LIN {X 0,Y 211.317,Z 790.887,A -85,B 0,C 180,E1 4630.049,E2 4630.049} C_VEL
LIN {X 0,Y 204.375,Z 802.097,A -85,B 0,C 180,E1 4624.722,E2 4624.722} C_VEL
LIN {X 0,Y 199.04,Z 811.282,A -85,B 0,C 180,E1 4619.061,E2 4619.061} C_VEL
LIN {X 0,Y 195.25,Z 818.98,A -85,B 0,C 180,E1 4612.9,E2 4612.9} C_VEL
LIN {X 0,Y 193.221,Z 824.706,A -85,B 0,C 180,E1 4606.795,E2 4606.795} C_VEL
LIN {X 0,Y 192.563,Z 828.46,A -85,B 0,C 180,E1 4601.073,E2 4601.073} C_VEL
LIN {X 0,Y 192.668,Z 830.823,A -85,B 0,C 180,E1 4595.357,E2 4595.357} C_VEL
LIN {X 0,Y 192.832,Z 831.611,A -85,B 0,C 180,E1 4590.591,E2 4590.591} C_VEL
LIN {X 0,Y 192.717,Z 831.408,A -85,B 0,C 180,E1 4586.13,E2 4586.13} C_VEL
LIN {X 0,Y 192.494,Z 830.016,A -85,B 0,C 180,E1 4580.727,E2 4580.727} C_VEL
LIN {X 0,Y 192.901,Z 826.886,A -85,B 0,C 180,E1 4574.669,E2 4574.669} C_VEL
LIN {X 0,Y 194.828,Z 821.744,A -85,B 0,C 180,E1 4567.995,E2 4567.995} C_VEL
LIN {X 0,Y 198.485,Z 815.132,A -85,B 0,C 180,E1 4561.734,E2 4561.734} C_VEL
LIN {X 0,Y 204.073,Z 806.598,A -85,B 0,C 180,E1 4555.703,E2 4555.703} C_VEL
LIN {X 0,Y 211.205,Z 796.698,A -85,B 0,C 180,E1 4550.272,E2 4550.272} C_VEL
LIN {X 0,Y 220.022,Z 784.872,A -85,B 0,C 180,E1 4545.218,E2 4545.218} C_VEL
LIN {X 0,Y 229.843,Z 771.631,A -85,B 0,C 180,E1 4540.802,E2 4540.802} C_VEL
LIN {X 0,Y 240.325,Z 756.815,A -85,B 0,C 180,E1 4536.981,E2 4536.981} C_VEL
LIN {X 0,Y 250.499,Z 741.511,A -85,B 0,C 180,E1 4533.875,E2 4533.875} C_VEL
LIN {X 0,Y 261.006,Z 724.467,A -85,B 0,C 180,E1 4531.143,E2 4531.143} C_VEL
LIN {X 0,Y 270.771,Z 707,A -85,B 0,C 180,E1 4528.931,E2 4528.931} C_VEL
LIN {X 0,Y 280.133,Z 688.021,A -85,B 0,C 180,E1 4527.058,E2 4527.058} C_VEL
LIN {X 0,Y 288.655,Z 668.181,A -85,B 0,C 180,E1 4525.53,E2 4525.53} C_VEL
LIN {X 0,Y 296.228,Z 647.353,A -85,B 0,C 180,E1 4524.307,E2 4524.307} C_VEL
LIN {X 0,Y 302.485,Z 626.505,A -85,B 0,C 180,E1 4523.392,E2 4523.392} C_VEL
LIN {X 0,Y 307.54,Z 604.237,A -85,B 0,C 180,E1 4522.67,E2 4522.67} C_VEL
LIN {X 0,Y 310.852,Z 582.325,A -85,B 0,C 180,E1 4522.123,E2 4522.123} C_VEL
LIN {X 0,Y 326.311,Z 437.595,A -85,B 0,C 180,E1 4519.094,E2 4519.094} C_VEL
LIN {X 0,Y 324.635,Z 433.151,A -85,B 0,C 180,E1 4517.015,E2 4517.015} C_VEL
LIN {X 0,Y 323.554,Z 430.422,A -85,B 0,C 180,E1 4515.23,E2 4515.23} C_VEL
LIN {X 0,Y 322.63,Z 427.763,A -85,B 0,C 180,E1 4512.712,E2 4512.712} C_VEL
LIN {X 0,Y 322.365,Z 427.503,A -85,B 0,C 180,E1 4509.103,E2 4509.103} C_VEL
LIN {X 0,Y 322.631,Z 428.25,A -85,B 0,C 180,E1 4507.749,E2 4507.749} C_VEL
LIN {X 0,Y 323.747,Z 431.704,A -85,B 0,C 180,E1 4504.873,E2 4504.873} C_VEL
LIN {X 0,Y 325.23,Z 435.825,A -85,B 0,C 180,E1 4502.645,E2 4502.645} C_VEL
LIN {X 0,Y 325.665,Z 437.428,A -85,B 0,C 180,E1 4502.072,E2 4502.072} C_VEL
LIN {X 0,Y 308.977,Z 582.418,A -85,B 0,C 180,E1 4499.021,E2 4499.021} C_VEL
LIN {X 0,Y 305.09,Z 603.307,A -85,B 0,C 180,E1 4498.354,E2 4498.354} C_VEL
LIN {X 0,Y 300.007,Z 623.447,A -85,B 0,C 180,E1 4497.469,E2 4497.469} C_VEL
LIN {X 0,Y 293.506,Z 643.814,A -85,B 0,C 180,E1 4496.291,E2 4496.291} C_VEL
LIN {X 0,Y 286.577,Z 661.874,A -85,B 0,C 180,E1 4494.957,E2 4494.957} C_VEL
LIN {X 0,Y 278.381,Z 679.801,A -85,B 0,C 180,E1 4493.278,E2 4493.278} C_VEL
LIN {X 0,Y 269.137,Z 697.434,A -85,B 0,C 180,E1 4491.201,E2 4491.201} C_VEL
LIN {X 0,Y 259.035,Z 714.421,A -85,B 0,C 180,E1 4488.653,E2 4488.653} C_VEL
LIN {X 0,Y 249.221,Z 729.24,A -85,B 0,C 180,E1 4485.836,E2 4485.836} C_VEL
LIN {X 0,Y 239.085,Z 743.194,A -85,B 0,C 180,E1 4482.465,E2 4482.465} C_VEL
LIN {X 0,Y 228.642,Z 756.385,A -85,B 0,C 180,E1 4478.327,E2 4478.327} C_VEL
LIN {X 0,Y 219.438,Z 767.23,A -85,B 0,C 180,E1 4473.852,E2 4473.852} C_VEL
LIN {X 0,Y 211.365,Z 776.379,A -85,B 0,C 180,E1 4468.899,E2 4468.899} C_VEL
LIN {X 0,Y 204.471,Z 784.06,A -85,B 0,C 180,E1 4463.321,E2 4463.321} C_VEL
LIN {X 0,Y 199.247,Z 789.969,A -85,B 0,C 180,E1 4457.359,E2 4457.359} C_VEL
LIN {X 0,Y 195.774,Z 794.085,A -85,B 0,C 180,E1 4451.214,E2 4451.214} C_VEL
LIN {X 0,Y 193.917,Z 796.385,A -85,B 0,C 180,E1 4445.277,E2 4445.277} C_VEL
LIN {X 0,Y 193.148,Z 797.233,A -85,B 0,C 180,E1 4439.461,E2 4439.461} C_VEL
LIN {X 0,Y 193.025,Z 796.836,A -85,B 0,C 180,E1 4433.834,E2 4433.834} C_VEL
LIN {X 0,Y 193.474,Z 794.978,A -85,B 0,C 180,E1 4428.041,E2 4428.041} C_VEL
LIN {X 0,Y 194.932,Z 791.439,A -85,B 0,C 180,E1 4421.843,E2 4421.843} C_VEL
LIN {X 0,Y 197.726,Z 786.247,A -85,B 0,C 180,E1 4415.808,E2 4415.808} C_VEL
LIN {X 0,Y 201.96,Z 779.409,A -85,B 0,C 180,E1 4410.063,E2 4410.063} C_VEL
LIN {X 0,Y 207.83,Z 770.496,A -85,B 0,C 180,E1 4404.481,E2 4404.481} C_VEL
LIN {X 0,Y 214.723,Z 760.117,A -85,B 0,C 180,E1 4399.54,E2 4399.54} C_VEL
LIN {X 0,Y 222.414,Z 748.305,A -85,B 0,C 180,E1 4395.156,E2 4395.156} C_VEL
LIN {X 0,Y 230.633,Z 735.088,A -85,B 0,C 180,E1 4391.291,E2 4391.291} C_VEL
LIN {X 0,Y 239.139,Z 720.459,A -85,B 0,C 180,E1 4387.898,E2 4387.898} C_VEL
LIN {X 0,Y 247.432,Z 704.923,A -85,B 0,C 180,E1 4385.024,E2 4385.024} C_VEL
LIN {X 0,Y 255.907,Z 687.184,A -85,B 0,C 180,E1 4382.423,E2 4382.423} C_VEL
LIN {X 0,Y 263.586,Z 668.825,A -85,B 0,C 180,E1 4380.298,E2 4380.298} C_VEL
LIN {X 0,Y 270.362,Z 650.051,A -85,B 0,C 180,E1 4378.573,E2 4378.573} C_VEL
LIN {X 0,Y 276.368,Z 630.229,A -85,B 0,C 180,E1 4377.137,E2 4377.137} C_VEL
LIN {X 0,Y 281.45,Z 609.5,A -85,B 0,C 180,E1 4375.988,E2 4375.988} C_VEL
LIN {X 0,Y 285.444,Z 588.089,A -85,B 0,C 180,E1 4375.117,E2 4375.117} C_VEL
LIN {X 0,Y 288.238,Z 565.56,A -85,B 0,C 180,E1 4374.491,E2 4374.491} C_VEL
LIN {X 0,Y 301.041,Z 423.363,A -85,B 0,C 180,E1 4371.364,E2 4371.364} C_VEL
LIN {X 0,Y 293.436,Z 409.422,A -85,B 0,C 180,E1 4367.547,E2 4367.547} C_VEL
LIN {X 0,Y 287.048,Z 398.81,A -85,B 0,C 180,E1 4363.864,E2 4363.864} C_VEL
LIN {X 0,Y 282.288,Z 391.221,A -85,B 0,C 180,E1 4360.669,E2 4360.669} C_VEL
LIN {X 0,Y 279.028,Z 386.353,A -85,B 0,C 180,E1 4358.177,E2 4358.177} C_VEL
LIN {X 0,Y 276.012,Z 381.873,A -85,B 0,C 180,E1 4355.547,E2 4355.547} C_VEL
LIN {X 0,Y 272.92,Z 377.285,A -85,B 0,C 180,E1 4352.333,E2 4352.333} C_VEL
LIN {X 0,Y 269.763,Z 372.7,A -85,B 0,C 180,E1 4348.078,E2 4348.078} C_VEL
LIN {X 0,Y 266.645,Z 368.098,A -85,B 0,C 180,E1 4340.637,E2 4340.637} C_VEL
LIN {X 0,Y 266.222,Z 367.692,A -85,B 0,C 180,E1 4334.572,E2 4334.572} C_VEL
LIN {X 0,Y 267.044,Z 368.731,A -85,B 0,C 180,E1 4330.57,E2 4330.57} C_VEL
LIN {X 0,Y 268.111,Z 370.684,A -85,B 0,C 180,E1 4327.627,E2 4327.627} C_VEL
LIN {X 0,Y 268.708,Z 372.408,A -85,B 0,C 180,E1 4326.259,E2 4326.259} C_VEL
LIN {X 0,Y 269.521,Z 377.466,A -85,B 0,C 180,E1 4324.137,E2 4324.137} C_VEL
LIN {X 0,Y 270.707,Z 383.214,A -85,B 0,C 180,E1 4321.82,E2 4321.82} C_VEL
LIN {X 0,Y 271.569,Z 384.888,A -85,B 0,C 180,E1 4320.705,E2 4320.705} C_VEL
LIN {X 0,Y 273.038,Z 386.963,A -85,B 0,C 180,E1 4319.065,E2 4319.065} C_VEL
LIN {X 0,Y 276.48,Z 392.054,A -85,B 0,C 180,E1 4315.747,E2 4315.747} C_VEL
LIN {X 0,Y 280.407,Z 397.981,A -85,B 0,C 180,E1 4312.572,E2 4312.572} C_VEL
LIN {X 0,Y 285.065,Z 405.319,A -85,B 0,C 180,E1 4309.336,E2 4309.336} C_VEL
LIN {X 0,Y 291.595,Z 415.977,A -85,B 0,C 180,E1 4305.452,E2 4305.452} C_VEL
LIN {X 0,Y 298.484,Z 428.22,A -85,B 0,C 180,E1 4301.898,E2 4301.898} C_VEL
LIN {X 0,Y 301.017,Z 433.158,A -85,B 0,C 180,E1 4300.693,E2 4300.693} C_VEL
LIN {X 0,Y 286.835,Z 594.303,A -85,B 0,C 180,E1 4297.252,E2 4297.252} C_VEL
LIN {X 0,Y 283.258,Z 616.443,A -85,B 0,C 180,E1 4296.578,E2 4296.578} C_VEL
LIN {X 0,Y 278.332,Z 637.822,A -85,B 0,C 180,E1 4295.714,E2 4295.714} C_VEL
LIN {X 0,Y 272.14,Z 659.139,A -85,B 0,C 180,E1 4294.54,E2 4294.54} C_VEL
LIN {X 0,Y 265.201,Z 679.03,A -85,B 0,C 180,E1 4293.099,E2 4293.099} C_VEL
LIN {X 0,Y 257.115,Z 698.659,A -85,B 0,C 180,E1 4291.266,E2 4291.266} C_VEL
LIN {X 0,Y 248.687,Z 716.603,A -85,B 0,C 180,E1 4289.13,E2 4289.13} C_VEL
LIN {X 0,Y 239.009,Z 735.048,A -85,B 0,C 180,E1 4286.349,E2 4286.349} C_VEL
LIN {X 0,Y 230.023,Z 750.696,A -85,B 0,C 180,E1 4283.358,E2 4283.358} C_VEL
LIN {X 0,Y 220.474,Z 766.1,A -85,B 0,C 180,E1 4279.626,E2 4279.626} C_VEL
LIN {X 0,Y 211.738,Z 779.481,A -85,B 0,C 180,E1 4275.478,E2 4275.478} C_VEL
LIN {X 0,Y 203.307,Z 792.156,A -85,B 0,C 180,E1 4270.475,E2 4270.475} C_VEL
LIN {X 0,Y 196.415,Z 802.743,A -85,B 0,C 180,E1 4265.112,E2 4265.112} C_VEL
LIN {X 0,Y 190.906,Z 811.872,A -85,B 0,C 180,E1 4259.145,E2 4259.145} C_VEL
LIN {X 0,Y 187.202,Z 819.025,A -85,B 0,C 180,E1 4252.944,E2 4252.944} C_VEL
LIN {X 0,Y 185.121,Z 824.711,A -85,B 0,C 180,E1 4246.308,E2 4246.308} C_VEL
LIN {X 0,Y 184.564,Z 828.324,A -85,B 0,C 180,E1 4240.295,E2 4240.295} C_VEL
LIN {X 0,Y 184.735,Z 830.276,A -85,B 0,C 180,E1 4234.653,E2 4234.653} C_VEL
LIN {X 0,Y 184.878,Z 830.91,A -85,B 0,C 180,E1 4229.997,E2 4229.997} C_VEL
LIN {X 0,Y 184.705,Z 830.615,A -85,B 0,C 180,E1 4225.339,E2 4225.339} C_VEL
LIN {X 0,Y 184.52,Z 828.929,A -85,B 0,C 180,E1 4219.38,E2 4219.38} C_VEL
LIN {X 0,Y 185.127,Z 825.839,A -85,B 0,C 180,E1 4213.363,E2 4213.363} C_VEL
LIN {X 0,Y 187.473,Z 820.555,A -85,B 0,C 180,E1 4206.418,E2 4206.418} C_VEL
LIN {X 0,Y 191.675,Z 813.79,A -85,B 0,C 180,E1 4199.945,E2 4199.945} C_VEL
LIN {X 0,Y 197.916,Z 805.198,A -85,B 0,C 180,E1 4193.763,E2 4193.763} C_VEL
LIN {X 0,Y 205.71,Z 795.146,A -85,B 0,C 180,E1 4188.246,E2 4188.246} C_VEL
LIN {X 0,Y 215.604,Z 782.696,A -85,B 0,C 180,E1 4182.979,E2 4182.979} C_VEL
LIN {X 0,Y 226.224,Z 769.059,A -85,B 0,C 180,E1 4178.551,E2 4178.551} C_VEL
LIN {X 0,Y 236.749,Z 754.9,A -85,B 0,C 180,E1 4174.98,E2 4174.98} C_VEL
LIN {X 0,Y 247.404,Z 739.443,A -85,B 0,C 180,E1 4171.926,E2 4171.926} C_VEL
LIN {X 0,Y 258.406,Z 722.059,A -85,B 0,C 180,E1 4169.242,E2 4169.242} C_VEL
LIN {X 0,Y 268.469,Z 704.499,A -85,B 0,C 180,E1 4167.11,E2 4167.11} C_VEL
LIN {X 0,Y 278.154,Z 685.338,A -85,B 0,C 180,E1 4165.301,E2 4165.301} C_VEL
LIN {X 0,Y 286.741,Z 665.592,A -85,B 0,C 180,E1 4163.86,E2 4163.86} C_VEL
LIN {X 0,Y 294.301,Z 645.023,A -85,B 0,C 180,E1 4162.718,E2 4162.718} C_VEL
LIN {X 0,Y 300.678,Z 623.698,A -85,B 0,C 180,E1 4161.842,E2 4161.842} C_VEL
LIN {X 0,Y 305.706,Z 601.598,A -85,B 0,C 180,E1 4161.161,E2 4161.161} C_VEL
LIN {X 0,Y 309.082,Z 578.98,A -85,B 0,C 180,E1 4160.621,E2 4160.621} C_VEL
LIN {X 0,Y 324.139,Z 443.084,A -85,B 0,C 180,E1 4157.844,E2 4157.844} C_VEL
LIN {X 0,Y 322.498,Z 438.528,A -85,B 0,C 180,E1 4155.281,E2 4155.281} C_VEL
LIN {X 0,Y 321.524,Z 435.658,A -85,B 0,C 180,E1 4152.574,E2 4152.574} C_VEL
LIN {X 0,Y 321.29,Z 435.43,A -85,B 0,C 180,E1 4149.134,E2 4149.134} C_VEL
LIN {X 0,Y 321.513,Z 436.195,A -85,B 0,C 180,E1 4147.866,E2 4147.866} C_VEL
LIN {X 0,Y 322.481,Z 439.462,A -85,B 0,C 180,E1 4145.16,E2 4145.16} C_VEL
LIN {X 0,Y 323.554,Z 442.72,A -85,B 0,C 180,E1 4143.358,E2 4143.358} C_VEL
LIN {X 0,Y 306.938,Z 582.808,A -85,B 0,C 180,E1 4140.461,E2 4140.461} C_VEL
LIN {X 0,Y 302.915,Z 603.797,A -85,B 0,C 180,E1 4139.806,E2 4139.806} C_VEL
LIN {X 0,Y 297.764,Z 623.721,A -85,B 0,C 180,E1 4138.954,E2 4138.954} C_VEL
LIN {X 0,Y 291.177,Z 643.893,A -85,B 0,C 180,E1 4137.82,E2 4137.82} C_VEL
LIN {X 0,Y 283.519,Z 663.131,A -85,B 0,C 180,E1 4136.423,E2 4136.423} C_VEL
LIN {X 0,Y 274.65,Z 681.852,A -85,B 0,C 180,E1 4134.684,E2 4134.684} C_VEL
LIN {X 0,Y 265.153,Z 699.145,A -85,B 0,C 180,E1 4132.643,E2 4132.643} C_VEL
LIN {X 0,Y 254.743,Z 715.871,A -85,B 0,C 180,E1 4130.129,E2 4130.129} C_VEL
LIN {X 0,Y 244.058,Z 731.223,A -85,B 0,C 180,E1 4127.18,E2 4127.18} C_VEL
LIN {X 0,Y 233.712,Z 744.734,A -85,B 0,C 180,E1 4123.857,E2 4123.857} C_VEL
LIN {X 0,Y 223.496,Z 757.002,A -85,B 0,C 180,E1 4119.971,E2 4119.971} C_VEL
LIN {X 0,Y 213.636,Z 768.004,A -85,B 0,C 180,E1 4115.387,E2 4115.387} C_VEL
LIN {X 0,Y 205.343,Z 776.816,A -85,B 0,C 180,E1 4110.545,E2 4110.545} C_VEL
LIN {X 0,Y 197.578,Z 784.879,A -85,B 0,C 180,E1 4104.567,E2 4104.567} C_VEL
LIN {X 0,Y 192.047,Z 790.635,A -85,B 0,C 180,E1 4098.569,E2 4098.569} C_VEL
LIN {X 0,Y 188.135,Z 794.847,A -85,B 0,C 180,E1 4092.043,E2 4092.043} C_VEL
LIN {X 0,Y 186.051,Z 797.16,A -85,B 0,C 180,E1 4085.764,E2 4085.764} C_VEL
LIN {X 0,Y 185.192,Z 797.967,A -85,B 0,C 180,E1 4079.636,E2 4079.636} C_VEL
LIN {X 0,Y 185.054,Z 797.56,A -85,B 0,C 180,E1 4073.909,E2 4073.909} C_VEL
LIN {X 0,Y 185.522,Z 795.705,A -85,B 0,C 180,E1 4067.894,E2 4067.894} C_VEL
LIN {X 0,Y 186.973,Z 792.374,A -85,B 0,C 180,E1 4061.728,E2 4061.728} C_VEL
LIN {X 0,Y 189.7,Z 787.592,A -85,B 0,C 180,E1 4055.751,E2 4055.751} C_VEL
LIN {X 0,Y 194.088,Z 780.826,A -85,B 0,C 180,E1 4049.708,E2 4049.708} C_VEL
LIN {X 0,Y 199.732,Z 772.618,A -85,B 0,C 180,E1 4044.257,E2 4044.257} C_VEL
LIN {X 0,Y 206.772,Z 762.571,A -85,B 0,C 180,E1 4039.133,E2 4039.133} C_VEL
LIN {X 0,Y 215.113,Z 750.424,A -85,B 0,C 180,E1 4034.363,E2 4034.363} C_VEL
LIN {X 0,Y 223.579,Z 737.487,A -85,B 0,C 180,E1 4030.406,E2 4030.406} C_VEL
LIN {X 0,Y 232.336,Z 723.177,A -85,B 0,C 180,E1 4026.948,E2 4026.948} C_VEL
LIN {X 0,Y 241.451,Z 706.786,A -85,B 0,C 180,E1 4023.834,E2 4023.834} C_VEL
LIN {X 0,Y 249.848,Z 689.894,A -85,B 0,C 180,E1 4021.303,E2 4021.303} C_VEL
LIN {X 0,Y 257.65,Z 672.182,A -85,B 0,C 180,E1 4019.189,E2 4019.189} C_VEL
LIN {X 0,Y 265.031,Z 652.803,A -85,B 0,C 180,E1 4017.355,E2 4017.355} C_VEL
LIN {X 0,Y 271.202,Z 633.569,A -85,B 0,C 180,E1 4015.92,E2 4015.92} C_VEL
LIN {X 0,Y 276.606,Z 612.831,A -85,B 0,C 180,E1 4014.731,E2 4014.731} C_VEL
LIN {X 0,Y 280.958,Z 590.736,A -85,B 0,C 180,E1 4013.808,E2 4013.808} C_VEL
LIN {X 0,Y 283.853,Z 569.055,A -85,B 0,C 180,E1 4013.186,E2 4013.186} C_VEL
LIN {X 0,Y 297.056,Z 427.726,A -85,B 0,C 180,E1 4010.119,E2 4010.119} C_VEL
LIN {X 0,Y 290.081,Z 414.776,A -85,B 0,C 180,E1 4006.424,E2 4006.424} C_VEL
LIN {X 0,Y 283.791,Z 404.153,A -85,B 0,C 180,E1 4002.564,E2 4002.564} C_VEL
LIN {X 0,Y 278.928,Z 396.293,A -85,B 0,C 180,E1 3999.041,E2 3999.041} C_VEL
LIN {X 0,Y 274.567,Z 389.623,A -85,B 0,C 180,E1 3995.25,E2 3995.25} C_VEL
LIN {X 0,Y 271.442,Z 384.916,A -85,B 0,C 180,E1 3991.907,E2 3991.907} C_VEL
LIN {X 0,Y 268.47,Z 380.465,A -85,B 0,C 180,E1 3987.742,E2 3987.742} C_VEL
LIN {X 0,Y 265.541,Z 375.997,A -85,B 0,C 180,E1 3980.496,E2 3980.496} C_VEL
LIN {X 0,Y 265.191,Z 375.642,A -85,B 0,C 180,E1 3974.321,E2 3974.321} C_VEL
LIN {X 0,Y 265.958,Z 376.69,A -85,B 0,C 180,E1 3970.613,E2 3970.613} C_VEL
LIN {X 0,Y 269.31,Z 381.434,A -85,B 0,C 180,E1 3963.723,E2 3963.723} C_VEL
LIN {X 0,Y 271.569,Z 384.888,A -85,B 0,C 180,E1 3960.705,E2 3960.705} C_VEL
LIN {X 0,Y 272.641,Z 387.183,A -85,B 0,C 180,E1 3959.412,E2 3959.412} C_VEL
LIN {X 0,Y 273.919,Z 392.722,A -85,B 0,C 180,E1 3957.666,E2 3957.666} C_VEL
LIN {X 0,Y 275.612,Z 399.966,A -85,B 0,C 180,E1 3955.586,E2 3955.586} C_VEL
LIN {X 0,Y 276.984,Z 402.781,A -85,B 0,C 180,E1 3954.35,E2 3954.35} C_VEL
LIN {X 0,Y 282.178,Z 411.083,A -85,B 0,C 180,E1 3950.463,E2 3950.463} C_VEL
LIN {X 0,Y 288.7,Z 422.062,A -85,B 0,C 180,E1 3946.377,E2 3946.377} C_VEL
LIN {X 0,Y 295.298,Z 433.977,A -85,B 0,C 180,E1 3942.816,E2 3942.816} C_VEL
LIN {X 0,Y 296.966,Z 437.33,A -85,B 0,C 180,E1 3941.97,E2 3941.97} C_VEL
LIN {X 0,Y 282.792,Z 593.873,A -85,B 0,C 180,E1 3938.648,E2 3938.648} C_VEL
LIN {X 0,Y 279.152,Z 615.981,A -85,B 0,C 180,E1 3937.982,E2 3937.982} C_VEL
LIN {X 0,Y 274.222,Z 637.006,A -85,B 0,C 180,E1 3937.149,E2 3937.149} C_VEL
LIN {X 0,Y 268.074,Z 657.865,A -85,B 0,C 180,E1 3936.028,E2 3936.028} C_VEL
LIN {X 0,Y 261.112,Z 677.502,A -85,B 0,C 180,E1 3934.642,E2 3934.642} C_VEL
LIN {X 0,Y 252.83,Z 697.157,A -85,B 0,C 180,E1 3932.842,E2 3932.842} C_VEL
LIN {X 0,Y 244.134,Z 715.263,A -85,B 0,C 180,E1 3930.726,E2 3930.726} C_VEL
LIN {X 0,Y 235.131,Z 732.09,A -85,B 0,C 180,E1 3928.257,E2 3928.257} C_VEL
LIN {X 0,Y 225.36,Z 748.711,A -85,B 0,C 180,E1 3925.159,E2 3925.159} C_VEL
LIN {X 0,Y 215.695,Z 763.753,A -85,B 0,C 180,E1 3921.568,E2 3921.568} C_VEL
LIN {X 0,Y 206.435,Z 777.433,A -85,B 0,C 180,E1 3917.404,E2 3917.404} C_VEL
LIN {X 0,Y 197.859,Z 789.749,A -85,B 0,C 180,E1 3912.617,E2 3912.617} C_VEL
LIN {X 0,Y 190.321,Z 800.653,A -85,B 0,C 180,E1 3907.164,E2 3907.164} C_VEL
LIN {X 0,Y 184.175,Z 809.989,A -85,B 0,C 180,E1 3901.043,E2 3901.043} C_VEL
LIN {X 0,Y 179.925,Z 817.446,A -85,B 0,C 180,E1 3894.628,E2 3894.628} C_VEL
LIN {X 0,Y 177.487,Z 823.186,A -85,B 0,C 180,E1 3888.046,E2 3888.046} C_VEL
LIN {X 0,Y 176.622,Z 827.046,A -85,B 0,C 180,E1 3881.655,E2 3881.655} C_VEL
LIN {X 0,Y 176.717,Z 829.379,A -85,B 0,C 180,E1 3875.516,E2 3875.516} C_VEL
LIN {X 0,Y 176.897,Z 830.15,A -85,B 0,C 180,E1 3870.644,E2 3870.644} C_VEL
LIN {X 0,Y 176.772,Z 830.023,A -85,B 0,C 180,E1 3866.105,E2 3866.105} C_VEL
LIN {X 0,Y 176.535,Z 828.911,A -85,B 0,C 180,E1 3860.872,E2 3860.872} C_VEL
LIN {X 0,Y 176.959,Z 826.121,A -85,B 0,C 180,E1 3854.26,E2 3854.26} C_VEL
LIN {X 0,Y 178.979,Z 821.599,A -85,B 0,C 180,E1 3847.324,E2 3847.324} C_VEL
LIN {X 0,Y 182.982,Z 815.305,A -85,B 0,C 180,E1 3840.539,E2 3840.539} C_VEL
LIN {X 0,Y 189.451,Z 806.849,A -85,B 0,C 180,E1 3833.762,E2 3833.762} C_VEL
LIN {X 0,Y 197.326,Z 797.426,A -85,B 0,C 180,E1 3828.018,E2 3828.018} C_VEL
LIN {X 0,Y 207.487,Z 785.453,A -85,B 0,C 180,E1 3822.495,E2 3822.495} C_VEL
LIN {X 0,Y 218.17,Z 772.52,A -85,B 0,C 180,E1 3817.973,E2 3817.973} C_VEL
LIN {X 0,Y 229.478,Z 758.232,A -85,B 0,C 180,E1 3814.118,E2 3814.118} C_VEL
LIN {X 0,Y 240.707,Z 743.031,A -85,B 0,C 180,E1 3810.929,E2 3810.929} C_VEL
LIN {X 0,Y 251.57,Z 727.055,A -85,B 0,C 180,E1 3808.312,E2 3808.312} C_VEL
LIN {X 0,Y 262.176,Z 709.638,A -85,B 0,C 180,E1 3806.084,E2 3806.084} C_VEL
LIN {X 0,Y 272.424,Z 690.815,A -85,B 0,C 180,E1 3804.206,E2 3804.206} C_VEL
LIN {X 0,Y 281.353,Z 672.019,A -85,B 0,C 180,E1 3802.747,E2 3802.747} C_VEL
LIN {X 0,Y 289.67,Z 651.339,A -85,B 0,C 180,E1 3801.524,E2 3801.524} C_VEL
LIN {X 0,Y 296.459,Z 630.741,A -85,B 0,C 180,E1 3800.62,E2 3800.62} C_VEL
LIN {X 0,Y 302.179,Z 608.48,A -85,B 0,C 180,E1 3799.893,E2 3799.893} C_VEL
LIN {X 0,Y 306.169,Z 586.363,A -85,B 0,C 180,E1 3799.333,E2 3799.333} C_VEL
LIN {X 0,Y 322.102,Z 448.808,A -85,B 0,C 180,E1 3796.549,E2 3796.549} C_VEL
LIN {X 0,Y 321.075,Z 445.855,A -85,B 0,C 180,E1 3794.611,E2 3794.611} C_VEL
LIN {X 0,Y 320.402,Z 443.533,A -85,B 0,C 180,E1 3792.371,E2 3792.371} C_VEL
LIN {X 0,Y 320.229,Z 443.404,A -85,B 0,C 180,E1 3788.983,E2 3788.983} C_VEL
LIN {X 0,Y 320.479,Z 444.647,A -85,B 0,C 180,E1 3787.531,E2 3787.531} C_VEL
LIN {X 0,Y 321.219,Z 447.217,A -85,B 0,C 180,E1 3785.449,E2 3785.449} C_VEL
LIN {X 0,Y 321.577,Z 448.718,A -85,B 0,C 180,E1 3784.649,E2 3784.649} C_VEL
LIN {X 0,Y 305.134,Z 583.368,A -85,B 0,C 180,E1 3781.917,E2 3781.917} C_VEL
LIN {X 0,Y 301.005,Z 604.432,A -85,B 0,C 180,E1 3781.277,E2 3781.277} C_VEL
LIN {X 0,Y 295.663,Z 624.495,A -85,B 0,C 180,E1 3780.44,E2 3780.44} C_VEL
LIN {X 0,Y 288.737,Z 644.962,A -85,B 0,C 180,E1 3779.313,E2 3779.313} C_VEL
LIN {X 0,Y 280.929,Z 663.951,A -85,B 0,C 180,E1 3777.962,E2 3777.962} C_VEL
LIN {X 0,Y 272.033,Z 682.159,A -85,B 0,C 180,E1 3776.31,E2 3776.31} C_VEL
LIN {X 0,Y 262.714,Z 698.621,A -85,B 0,C 180,E1 3774.422,E2 3774.422} C_VEL
LIN {X 0,Y 252.176,Z 715.162,A -85,B 0,C 180,E1 3772.025,E2 3772.025} C_VEL
LIN {X 0,Y 241.492,Z 730.093,A -85,B 0,C 180,E1 3769.264,E2 3769.264} C_VEL
LIN {X 0,Y 230.394,Z 744.103,A -85,B 0,C 180,E1 3765.937,E2 3765.937} C_VEL
LIN {X 0,Y 219.604,Z 756.455,A -85,B 0,C 180,E1 3762.103,E2 3762.103} C_VEL
LIN {X 0,Y 209.558,Z 767.177,A -85,B 0,C 180,E1 3757.769,E2 3757.769} C_VEL
LIN {X 0,Y 200.053,Z 776.749,A -85,B 0,C 180,E1 3752.628,E2 3752.628} C_VEL
LIN {X 0,Y 192.04,Z 784.547,A -85,B 0,C 180,E1 3746.961,E2 3746.961} C_VEL
LIN {X 0,Y 185.732,Z 790.596,A -85,B 0,C 180,E1 3740.828,E2 3740.828} C_VEL
LIN {X 0,Y 181.149,Z 794.99,A -85,B 0,C 180,E1 3734.153,E2 3734.153} C_VEL
LIN {X 0,Y 178.538,Z 797.565,A -85,B 0,C 180,E1 3727.624,E2 3727.624} C_VEL
LIN {X 0,Y 177.344,Z 798.688,A -85,B 0,C 180,E1 3721.029,E2 3721.029} C_VEL
LIN {X 0,Y 177.065,Z 798.448,A -85,B 0,C 180,E1 3715.387,E2 3715.387} C_VEL
LIN {X 0,Y 177.397,Z 796.935,A -85,B 0,C 180,E1 3709.084,E2 3709.084} C_VEL
LIN {X 0,Y 178.698,Z 793.961,A -85,B 0,C 180,E1 3702.607,E2 3702.607} C_VEL
LIN {X 0,Y 181.482,Z 789.142,A -85,B 0,C 180,E1 3696.012,E2 3696.012} C_VEL
LIN {X 0,Y 185.633,Z 782.975,A -85,B 0,C 180,E1 3690.003,E2 3690.003} C_VEL
LIN {X 0,Y 191.637,Z 774.71,A -85,B 0,C 180,E1 3684.014,E2 3684.014} C_VEL
LIN {X 0,Y 198.829,Z 764.999,A -85,B 0,C 180,E1 3678.693,E2 3678.693} C_VEL
LIN {X 0,Y 207.045,Z 753.711,A -85,B 0,C 180,E1 3673.936,E2 3673.936} C_VEL
LIN {X 0,Y 216.04,Z 740.65,A -85,B 0,C 180,E1 3669.693,E2 3669.693} C_VEL
LIN {X 0,Y 224.996,Z 726.678,A -85,B 0,C 180,E1 3666.15,E2 3666.15} C_VEL
LIN {X 0,Y 234.014,Z 711.36,A -85,B 0,C 180,E1 3663.073,E2 3663.073} C_VEL
LIN {X 0,Y 242.908,Z 694.571,A -85,B 0,C 180,E1 3660.403,E2 3660.403} C_VEL
LIN {X 0,Y 251.066,Z 677.263,A -85,B 0,C 180,E1 3658.218,E2 3658.218} C_VEL
LIN {X 0,Y 258.777,Z 658.321,A -85,B 0,C 180,E1 3656.33,E2 3656.33} C_VEL
LIN {X 0,Y 265.436,Z 638.871,A -85,B 0,C 180,E1 3654.811,E2 3654.811} C_VEL
LIN {X 0,Y 271.137,Z 618.576,A -85,B 0,C 180,E1 3653.582,E2 3653.582} C_VEL
LIN {X 0,Y 275.928,Z 596.61,A -85,B 0,C 180,E1 3652.593,E2 3652.593} C_VEL
LIN {X 0,Y 279.265,Z 575.086,A -85,B 0,C 180,E1 3651.911,E2 3651.911} C_VEL
LIN {X 0,Y 293.087,Z 431.982,A -85,B 0,C 180,E1 3648.795,E2 3648.795} C_VEL
LIN {X 0,Y 287.064,Z 420.653,A -85,B 0,C 180,E1 3645.418,E2 3645.418} C_VEL
LIN {X 0,Y 281.27,Z 410.507,A -85,B 0,C 180,E1 3641.66,E2 3641.66} C_VEL
LIN {X 0,Y 276.296,Z 402.274,A -85,B 0,C 180,E1 3637.832,E2 3637.832} C_VEL
LIN {X 0,Y 272.793,Z 396.922,A -85,B 0,C 180,E1 3634.616,E2 3634.616} C_VEL
LIN {X 0,Y 270.117,Z 392.708,A -85,B 0,C 180,E1 3631.645,E2 3631.645} C_VEL
LIN {X 0,Y 267.258,Z 388.321,A -85,B 0,C 180,E1 3627.55,E2 3627.55} C_VEL
LIN {X 0,Y 264.435,Z 383.892,A -85,B 0,C 180,E1 3620.337,E2 3620.337} C_VEL
LIN {X 0,Y 264.138,Z 383.578,A -85,B 0,C 180,E1 3614.242,E2 3614.242} C_VEL
LIN {X 0,Y 264.807,Z 384.515,A -85,B 0,C 180,E1 3610.88,E2 3610.88} C_VEL
LIN {X 0,Y 268.055,Z 389.309,A -85,B 0,C 180,E1 3603.955,E2 3603.955} C_VEL
LIN {X 0,Y 271.463,Z 394.422,A -85,B 0,C 180,E1 3599.576,E2 3599.576} C_VEL
LIN {X 0,Y 274.903,Z 399.693,A -85,B 0,C 180,E1 3596.14,E2 3596.14} C_VEL
LIN {X 0,Y 276.984,Z 402.781,A -85,B 0,C 180,E1 3594.35,E2 3594.35} C_VEL
LIN {X 0,Y 278.417,Z 405.687,A -85,B 0,C 180,E1 3593.158,E2 3593.158} C_VEL
LIN {X 0,Y 280.067,Z 412.086,A -85,B 0,C 180,E1 3591.605,E2 3591.605} C_VEL
LIN {X 0,Y 282.309,Z 421.276,A -85,B 0,C 180,E1 3589.615,E2 3589.615} C_VEL
LIN {X 0,Y 283.62,Z 424.312,A -85,B 0,C 180,E1 3588.691,E2 3588.691} C_VEL
LIN {X 0,Y 288.994,Z 433.849,A -85,B 0,C 180,E1 3585.472,E2 3585.472} C_VEL
LIN {X 0,Y 293.045,Z 441.673,A -85,B 0,C 180,E1 3583.278,E2 3583.278} C_VEL
LIN {X 0,Y 278.869,Z 593.532,A -85,B 0,C 180,E1 3580.077,E2 3580.077} C_VEL
LIN {X 0,Y 275.139,Z 615.665,A -85,B 0,C 180,E1 3579.417,E2 3579.417} C_VEL
LIN {X 0,Y 270.081,Z 636.741,A -85,B 0,C 180,E1 3578.594,E2 3578.594} C_VEL
LIN {X 0,Y 263.595,Z 658.125,A -85,B 0,C 180,E1 3577.456,E2 3577.456} C_VEL
LIN {X 0,Y 256.407,Z 677.808,A -85,B 0,C 180,E1 3576.073,E2 3576.073} C_VEL
LIN {X 0,Y 247.983,Z 697.255,A -85,B 0,C 180,E1 3574.302,E2 3574.302} C_VEL
LIN {X 0,Y 239.05,Z 715.283,A -85,B 0,C 180,E1 3572.199,E2 3572.199} C_VEL
LIN {X 0,Y 229.139,Z 733.11,A -85,B 0,C 180,E1 3569.551,E2 3569.551} C_VEL
LIN {X 0,Y 219.36,Z 749.085,A -85,B 0,C 180,E1 3566.519,E2 3566.519} C_VEL
LIN {X 0,Y 209.37,Z 764.013,A -85,B 0,C 180,E1 3562.888,E2 3562.888} C_VEL
LIN {X 0,Y 199.726,Z 777.606,A -85,B 0,C 180,E1 3558.636,E2 3558.636} C_VEL
LIN {X 0,Y 190.379,Z 790.367,A -85,B 0,C 180,E1 3553.467,E2 3553.467} C_VEL
LIN {X 0,Y 182.59,Z 801.059,A -85,B 0,C 180,E1 3547.825,E2 3547.825} C_VEL
LIN {X 0,Y 176.247,Z 810.241,A -85,B 0,C 180,E1 3541.457,E2 3541.457} C_VEL
LIN {X 0,Y 171.885,Z 817.467,A -85,B 0,C 180,E1 3534.756,E2 3534.756} C_VEL
LIN {X 0,Y 169.358,Z 823.209,A -85,B 0,C 180,E1 3527.519,E2 3527.519} C_VEL
LIN {X 0,Y 168.618,Z 826.847,A -85,B 0,C 180,E1 3520.934,E2 3520.934} C_VEL
LIN {X 0,Y 168.79,Z 828.826,A -85,B 0,C 180,E1 3514.753,E2 3514.753} C_VEL
LIN {X 0,Y 168.944,Z 829.445,A -85,B 0,C 180,E1 3509.996,E2 3509.996} C_VEL
LIN {X 0,Y 168.754,Z 829.229,A -85,B 0,C 180,E1 3505.238,E2 3505.238} C_VEL
LIN {X 0,Y 168.555,Z 827.839,A -85,B 0,C 180,E1 3499.054,E2 3499.054} C_VEL
LIN {X 0,Y 169.372,Z 824.711,A -85,B 0,C 180,E1 3492.12,E2 3492.12} C_VEL
LIN {X 0,Y 172.222,Z 819.624,A -85,B 0,C 180,E1 3484.553,E2 3484.553} C_VEL
LIN {X 0,Y 177.159,Z 813.059,A -85,B 0,C 180,E1 3477.573,E2 3477.573} C_VEL
LIN {X 0,Y 184.321,Z 804.625,A -85,B 0,C 180,E1 3471.002,E2 3471.002} C_VEL
LIN {X 0,Y 193.595,Z 794.318,A -85,B 0,C 180,E1 3464.959,E2 3464.959} C_VEL
LIN {X 0,Y 204.206,Z 782.559,A -85,B 0,C 180,E1 3459.757,E2 3459.757} C_VEL
LIN {X 0,Y 215.719,Z 769.419,A -85,B 0,C 180,E1 3455.334,E2 3455.334} C_VEL
LIN {X 0,Y 227.725,Z 754.719,A -85,B 0,C 180,E1 3451.59,E2 3451.59} C_VEL
LIN {X 0,Y 239.541,Z 739.072,A -85,B 0,C 180,E1 3448.517,E2 3448.517} C_VEL
LIN {X 0,Y 251.668,Z 721.426,A -85,B 0,C 180,E1 3445.855,E2 3445.855} C_VEL
LIN {X 0,Y 262.374,Z 704.043,A -85,B 0,C 180,E1 3443.827,E2 3443.827} C_VEL
LIN {X 0,Y 272.963,Z 684.401,A -85,B 0,C 180,E1 3442.064,E2 3442.064} C_VEL
LIN {X 0,Y 281.752,Z 665.375,A -85,B 0,C 180,E1 3440.753,E2 3440.753} C_VEL
LIN {X 0,Y 289.876,Z 644.546,A -85,B 0,C 180,E1 3439.666,E2 3439.666} C_VEL
LIN {X 0,Y 296.546,Z 623.644,A -85,B 0,C 180,E1 3438.861,E2 3438.861} C_VEL
LIN {X 0,Y 301.936,Z 601.356,A -85,B 0,C 180,E1 3438.212,E2 3438.212} C_VEL
LIN {X 0,Y 305.551,Z 578.732,A -85,B 0,C 180,E1 3437.697,E2 3437.697} C_VEL
LIN {X 0,Y 320.263,Z 454.862,A -85,B 0,C 180,E1 3435.246,E2 3435.246} C_VEL
LIN {X 0,Y 319.31,Z 451.447,A -85,B 0,C 180,E1 3432.295,E2 3432.295} C_VEL
LIN {X 0,Y 319.147,Z 451.332,A -85,B 0,C 180,E1 3429.014,E2 3429.014} C_VEL
LIN {X 0,Y 319.863,Z 454.51,A -85,B 0,C 180,E1 3426.012,E2 3426.012} C_VEL
LIN {X 0,Y 319.672,Z 456.27,A -85,B 0,C 180,E1 3425.929,E2 3425.929} C_VEL
LIN {X 0,Y 303.625,Z 584.041,A -85,B 0,C 180,E1 3423.39,E2 3423.39} C_VEL
LIN {X 0,Y 299.356,Z 605.151,A -85,B 0,C 180,E1 3422.766,E2 3422.766} C_VEL
LIN {X 0,Y 293.836,Z 625.236,A -85,B 0,C 180,E1 3421.952,E2 3421.952} C_VEL
LIN {X 0,Y 286.685,Z 645.748,A -85,B 0,C 180,E1 3420.852,E2 3420.852} C_VEL
LIN {X 0,Y 278.975,Z 664.066,A -85,B 0,C 180,E1 3419.591,E2 3419.591} C_VEL
LIN {X 0,Y 270.125,Z 681.653,A -85,B 0,C 180,E1 3418.051,E2 3418.051} C_VEL
LIN {X 0,Y 260.065,Z 699.035,A -85,B 0,C 180,E1 3416.125,E2 3416.125} C_VEL
LIN {X 0,Y 249.148,Z 715.579,A -85,B 0,C 180,E1 3413.782,E2 3413.782} C_VEL
LIN {X 0,Y 237.887,Z 730.759,A -85,B 0,C 180,E1 3411.025,E2 3411.025} C_VEL
LIN {X 0,Y 226.173,Z 744.893,A -85,B 0,C 180,E1 3407.694,E2 3407.694} C_VEL
LIN {X 0,Y 214.6,Z 757.537,A -85,B 0,C 180,E1 3403.769,E2 3403.769} C_VEL
LIN {X 0,Y 203.846,Z 768.346,A -85,B 0,C 180,E1 3399.322,E2 3399.322} C_VEL
LIN {X 0,Y 193.583,Z 778.047,A -85,B 0,C 180,E1 3393.961,E2 3393.961} C_VEL
LIN {X 0,Y 184.93,Z 785.843,A -85,B 0,C 180,E1 3388.008,E2 3388.008} C_VEL
LIN {X 0,Y 178.32,Z 791.705,A -85,B 0,C 180,E1 3381.725,E2 3381.725} C_VEL
LIN {X 0,Y 173.403,Z 796.026,A -85,B 0,C 180,E1 3374.71,E2 3374.71} C_VEL
LIN {X 0,Y 170.574,Z 798.505,A -85,B 0,C 180,E1 3367.696,E2 3367.696} C_VEL
LIN {X 0,Y 169.361,Z 799.43,A -85,B 0,C 180,E1 3360.909,E2 3360.909} C_VEL
LIN {X 0,Y 169.099,Z 799.093,A -85,B 0,C 180,E1 3354.826,E2 3354.826} C_VEL
LIN {X 0,Y 169.527,Z 797.384,A -85,B 0,C 180,E1 3348.219,E2 3348.219} C_VEL
LIN {X 0,Y 171.052,Z 794.224,A -85,B 0,C 180,E1 3341.467,E2 3341.467} C_VEL
LIN {X 0,Y 174.205,Z 789.3,A -85,B 0,C 180,E1 3334.612,E2 3334.612} C_VEL
LIN {X 0,Y 179.082,Z 782.575,A -85,B 0,C 180,E1 3328.084,E2 3328.084} C_VEL
LIN {X 0,Y 185.327,Z 774.462,A -85,B 0,C 180,E1 3322.252,E2 3322.252} C_VEL
LIN {X 0,Y 193.061,Z 764.518,A -85,B 0,C 180,E1 3316.831,E2 3316.831} C_VEL
LIN {X 0,Y 201.644,Z 753.191,A -85,B 0,C 180,E1 3312.099,E2 3312.099} C_VEL
LIN {X 0,Y 210.751,Z 740.518,A -85,B 0,C 180,E1 3307.992,E2 3307.992} C_VEL
LIN {X 0,Y 220.106,Z 726.387,A -85,B 0,C 180,E1 3304.437,E2 3304.437} C_VEL
LIN {X 0,Y 229.482,Z 710.876,A -85,B 0,C 180,E1 3301.365,E2 3301.365} C_VEL
LIN {X 0,Y 238.704,Z 693.869,A -85,B 0,C 180,E1 3298.712,E2 3298.712} C_VEL
LIN {X 0,Y 247.3,Z 675.914,A -85,B 0,C 180,E1 3296.507,E2 3296.507} C_VEL
LIN {X 0,Y 255.089,Z 657.109,A -85,B 0,C 180,E1 3294.683,E2 3294.683} C_VEL
LIN {X 0,Y 261.944,Z 637.326,A -85,B 0,C 180,E1 3293.185,E2 3293.185} C_VEL
LIN {X 0,Y 267.614,Z 617.161,A -85,B 0,C 180,E1 3292.012,E2 3292.012} C_VEL
LIN {X 0,Y 272.296,Z 595.728,A -85,B 0,C 180,E1 3291.082,E2 3291.082} C_VEL
LIN {X 0,Y 275.78,Z 572.919,A -85,B 0,C 180,E1 3290.395,E2 3290.395} C_VEL
LIN {X 0,Y 289.263,Z 436.335,A -85,B 0,C 180,E1 3287.453,E2 3287.453} C_VEL
LIN {X 0,Y 284.362,Z 426.934,A -85,B 0,C 180,E1 3284.542,E2 3284.542} C_VEL
LIN {X 0,Y 278.637,Z 416.589,A -85,B 0,C 180,E1 3280.636,E2 3280.636} C_VEL
LIN {X 0,Y 273.882,Z 408.798,A -85,B 0,C 180,E1 3276.775,E2 3276.775} C_VEL
LIN {X 0,Y 271.128,Z 404.367,A -85,B 0,C 180,E1 3274.091,E2 3274.091} C_VEL
LIN {X 0,Y 268.611,Z 400.283,A -85,B 0,C 180,E1 3271.156,E2 3271.156} C_VEL
LIN {X 0,Y 266.009,Z 396.137,A -85,B 0,C 180,E1 3267.292,E2 3267.292} C_VEL
LIN {X 0,Y 263.338,Z 391.797,A -85,B 0,C 180,E1 3260.211,E2 3260.211} C_VEL
LIN {X 0,Y 263.1,Z 391.522,A -85,B 0,C 180,E1 3254.075,E2 3254.075} C_VEL
LIN {X 0,Y 263.724,Z 392.477,A -85,B 0,C 180,E1 3250.919,E2 3250.919} C_VEL
LIN {X 0,Y 266.739,Z 397.043,A -85,B 0,C 180,E1 3244.298,E2 3244.298} C_VEL
LIN {X 0,Y 269.981,Z 402.031,A -85,B 0,C 180,E1 3239.998,E2 3239.998} C_VEL
LIN {X 0,Y 273.337,Z 407.329,A -85,B 0,C 180,E1 3236.538,E2 3236.538} C_VEL
LIN {X 0,Y 277.176,Z 413.394,A -85,B 0,C 180,E1 3233.266,E2 3233.266} C_VEL
LIN {X 0,Y 281.678,Z 420.935,A -85,B 0,C 180,E1 3229.982,E2 3229.982} C_VEL
LIN {X 0,Y 283.62,Z 424.312,A -85,B 0,C 180,E1 3228.691,E2 3228.691} C_VEL
LIN {X 0,Y 284.711,Z 427.592,A -85,B 0,C 180,E1 3227.906,E2 3227.906} C_VEL
LIN {X 0,Y 286.587,Z 440.007,A -85,B 0,C 180,E1 3226.172,E2 3226.172} C_VEL
LIN {X 0,Y 287.459,Z 442.376,A -85,B 0,C 180,E1 3225.615,E2 3225.615} C_VEL
LIN {X 0,Y 289.204,Z 446.015,A -85,B 0,C 180,E1 3224.614,E2 3224.614} C_VEL
LIN {X 0,Y 275.102,Z 593.187,A -85,B 0,C 180,E1 3221.542,E2 3221.542} C_VEL
LIN {X 0,Y 271.275,Z 615.415,A -85,B 0,C 180,E1 3220.89,E2 3220.89} C_VEL
LIN {X 0,Y 266.118,Z 636.456,A -85,B 0,C 180,E1 3220.084,E2 3220.084} C_VEL
LIN {X 0,Y 259.697,Z 657.218,A -85,B 0,C 180,E1 3219.003,E2 3219.003} C_VEL
LIN {X 0,Y 252.273,Z 677.117,A -85,B 0,C 180,E1 3217.635,E2 3217.635} C_VEL
LIN {X 0,Y 243.692,Z 696.445,A -85,B 0,C 180,E1 3215.903,E2 3215.903} C_VEL
LIN {X 0,Y 234.504,Z 714.517,A -85,B 0,C 180,E1 3213.826,E2 3213.826} C_VEL
LIN {X 0,Y 224.412,Z 732.17,A -85,B 0,C 180,E1 3211.235,E2 3211.235} C_VEL
LIN {X 0,Y 214.16,Z 748.41,A -85,B 0,C 180,E1 3208.174,E2 3208.174} C_VEL
LIN {X 0,Y 203.785,Z 763.375,A -85,B 0,C 180,E1 3204.529,E2 3204.529} C_VEL
LIN {X 0,Y 193.745,Z 776.925,A -85,B 0,C 180,E1 3200.254,E2 3200.254} C_VEL
LIN {X 0,Y 183.891,Z 789.732,A -85,B 0,C 180,E1 3194.973,E2 3194.973} C_VEL
LIN {X 0,Y 175.651,Z 800.426,A -85,B 0,C 180,E1 3189.181,E2 3189.181} C_VEL
LIN {X 0,Y 168.892,Z 809.619,A -85,B 0,C 180,E1 3182.593,E2 3182.593} C_VEL
LIN {X 0,Y 164.206,Z 816.834,A -85,B 0,C 180,E1 3175.611,E2 3175.611} C_VEL
LIN {X 0,Y 161.461,Z 822.556,A -85,B 0,C 180,E1 3168.033,E2 3168.033} C_VEL
LIN {X 0,Y 160.643,Z 826.179,A -85,B 0,C 180,E1 3161.121,E2 3161.121} C_VEL
LIN {X 0,Y 160.826,Z 828.131,A -85,B 0,C 180,E1 3154.632,E2 3154.632} C_VEL
LIN {X 0,Y 160.967,Z 828.724,A -85,B 0,C 180,E1 3149.64,E2 3149.64} C_VEL
LIN {X 0,Y 160.733,Z 828.45,A -85,B 0,C 180,E1 3144.463,E2 3144.463} C_VEL
LIN {X 0,Y 160.614,Z 826.908,A -85,B 0,C 180,E1 3137.777,E2 3137.777} C_VEL
LIN {X 0,Y 161.755,Z 823.687,A -85,B 0,C 180,E1 3130.497,E2 3130.497} C_VEL
LIN {X 0,Y 165.404,Z 818.178,A -85,B 0,C 180,E1 3122.256,E2 3122.256} C_VEL
LIN {X 0,Y 171.148,Z 811.425,A -85,B 0,C 180,E1 3115.07,E2 3115.07} C_VEL
LIN {X 0,Y 179.636,Z 802.42,A -85,B 0,C 180,E1 3108.089,E2 3108.089} C_VEL
LIN {X 0,Y 189.371,Z 792.318,A -85,B 0,C 180,E1 3102.334,E2 3102.334} C_VEL
LIN {X 0,Y 200.821,Z 780.353,A -85,B 0,C 180,E1 3097.188,E2 3097.188} C_VEL
LIN {X 0,Y 213.061,Z 766.96,A -85,B 0,C 180,E1 3092.854,E2 3092.854} C_VEL
LIN {X 0,Y 225.71,Z 752.127,A -85,B 0,C 180,E1 3089.224,E2 3089.224} C_VEL
LIN {X 0,Y 238.066,Z 736.211,A -85,B 0,C 180,E1 3086.27,E2 3086.27} C_VEL
LIN {X 0,Y 249.856,Z 719.401,A -85,B 0,C 180,E1 3083.875,E2 3083.875} C_VEL
LIN {X 0,Y 260.864,Z 701.915,A -85,B 0,C 180,E1 3081.939,E2 3081.939} C_VEL
LIN {X 0,Y 270.926,Z 683.683,A -85,B 0,C 180,E1 3080.377,E2 3080.377} C_VEL
LIN {X 0,Y 279.918,Z 664.748,A -85,B 0,C 180,E1 3079.124,E2 3079.124} C_VEL
LIN {X 0,Y 288.213,Z 644.041,A -85,B 0,C 180,E1 3078.089,E2 3078.089} C_VEL
LIN {X 0,Y 295.004,Z 623.157,A -85,B 0,C 180,E1 3077.323,E2 3077.323} C_VEL
LIN {X 0,Y 300.545,Z 600.801,A -85,B 0,C 180,E1 3076.698,E2 3076.698} C_VEL
LIN {X 0,Y 304.293,Z 578.052,A -85,B 0,C 180,E1 3076.196,E2 3076.196} C_VEL
LIN {X 0,Y 318.631,Z 461.245,A -85,B 0,C 180,E1 3073.942,E2 3073.942} C_VEL
LIN {X 0,Y 318.168,Z 459.293,A -85,B 0,C 180,E1 3071.972,E2 3071.972} C_VEL
LIN {X 0,Y 318.085,Z 459.321,A -85,B 0,C 180,E1 3068.862,E2 3068.862} C_VEL
LIN {X 0,Y 318.305,Z 461.308,A -85,B 0,C 180,E1 3067.271,E2 3067.271} C_VEL
LIN {X 0,Y 302.419,Z 584.504,A -85,B 0,C 180,E1 3064.885,E2 3064.885} C_VEL
LIN {X 0,Y 298.048,Z 605.559,A -85,B 0,C 180,E1 3064.284,E2 3064.284} C_VEL
LIN {X 0,Y 292.254,Z 626.111,A -85,B 0,C 180,E1 3063.478,E2 3063.478} C_VEL
LIN {X 0,Y 284.926,Z 646.575,A -85,B 0,C 180,E1 3062.415,E2 3062.415} C_VEL
LIN {X 0,Y 276.521,Z 665.768,A -85,B 0,C 180,E1 3061.122,E2 3061.122} C_VEL
LIN {X 0,Y 266.978,Z 684.092,A -85,B 0,C 180,E1 3059.54,E2 3059.54} C_VEL
LIN {X 0,Y 256.684,Z 701.063,A -85,B 0,C 180,E1 3057.669,E2 3057.669} C_VEL
LIN {X 0,Y 245.215,Z 717.646,A -85,B 0,C 180,E1 3055.324,E2 3055.324} C_VEL
LIN {X 0,Y 233.681,Z 732.467,A -85,B 0,C 180,E1 3052.627,E2 3052.627} C_VEL
LIN {X 0,Y 221.609,Z 746.381,A -85,B 0,C 180,E1 3049.342,E2 3049.342} C_VEL
LIN {X 0,Y 209.683,Z 758.755,A -85,B 0,C 180,E1 3045.473,E2 3045.473} C_VEL
LIN {X 0,Y 198.667,Z 769.229,A -85,B 0,C 180,E1 3041.123,E2 3041.123} C_VEL
LIN {X 0,Y 188.002,Z 778.688,A -85,B 0,C 180,E1 3035.829,E2 3035.829} C_VEL
LIN {X 0,Y 178.996,Z 786.285,A -85,B 0,C 180,E1 3029.982,E2 3029.982} C_VEL
LIN {X 0,Y 171.683,Z 792.248,A -85,B 0,C 180,E1 3023.489,E2 3023.489} C_VEL
LIN {X 0,Y 166.182,Z 796.613,A -85,B 0,C 180,E1 3016.223,E2 3016.223} C_VEL
LIN {X 0,Y 163.022,Z 799.091,A -85,B 0,C 180,E1 3009.182,E2 3009.182} C_VEL
LIN {X 0,Y 161.511,Z 800.164,A -85,B 0,C 180,E1 3001.999,E2 3001.999} C_VEL
LIN {X 0,Y 161.127,Z 799.897,A -85,B 0,C 180,E1 2995.75,E2 2995.75} C_VEL
LIN {X 0,Y 161.485,Z 798.349,A -85,B 0,C 180,E1 2988.786,E2 2988.786} C_VEL
LIN {X 0,Y 162.975,Z 795.356,A -85,B 0,C 180,E1 2981.684,E2 2981.684} C_VEL
LIN {X 0,Y 166.169,Z 790.521,A -85,B 0,C 180,E1 2974.49,E2 2974.49} C_VEL
LIN {X 0,Y 171.096,Z 784.084,A -85,B 0,C 180,E1 2967.76,E2 2967.76} C_VEL
LIN {X 0,Y 178.024,Z 775.588,A -85,B 0,C 180,E1 2961.281,E2 2961.281} C_VEL
LIN {X 0,Y 186.098,Z 765.746,A -85,B 0,C 180,E1 2955.695,E2 2955.695} C_VEL
LIN {X 0,Y 195.034,Z 754.535,A -85,B 0,C 180,E1 2950.85,E2 2950.85} C_VEL
LIN {X 0,Y 205.064,Z 741.148,A -85,B 0,C 180,E1 2946.437,E2 2946.437} C_VEL
LIN {X 0,Y 214.786,Z 727.01,A -85,B 0,C 180,E1 2942.861,E2 2942.861} C_VEL
LIN {X 0,Y 224.496,Z 711.497,A -85,B 0,C 180,E1 2939.786,E2 2939.786} C_VEL
LIN {X 0,Y 234.02,Z 694.479,A -85,B 0,C 180,E1 2937.142,E2 2937.142} C_VEL
LIN {X 0,Y 242.871,Z 676.511,A -85,B 0,C 180,E1 2934.953,E2 2934.953} C_VEL
LIN {X 0,Y 250.876,Z 657.696,A -85,B 0,C 180,E1 2933.147,E2 2933.147} C_VEL
LIN {X 0,Y 257.91,Z 637.896,A -85,B 0,C 180,E1 2931.667,E2 2931.667} C_VEL
LIN {X 0,Y 263.723,Z 617.732,A -85,B 0,C 180,E1 2930.51,E2 2930.51} C_VEL
LIN {X 0,Y 268.543,Z 596.199,A -85,B 0,C 180,E1 2929.589,E2 2929.589} C_VEL
LIN {X 0,Y 272.11,Z 573.404,A -85,B 0,C 180,E1 2928.912,E2 2928.912} C_VEL
LIN {X 0,Y 285.574,Z 440.733,A -85,B 0,C 180,E1 2926.09,E2 2926.09} C_VEL
LIN {X 0,Y 280.642,Z 431.184,A -85,B 0,C 180,E1 2922.948,E2 2922.948} C_VEL
LIN {X 0,Y 275.33,Z 421.526,A -85,B 0,C 180,E1 2919.005,E2 2919.005} C_VEL
LIN {X 0,Y 271.801,Z 415.656,A -85,B 0,C 180,E1 2915.924,E2 2915.924} C_VEL
LIN {X 0,Y 269.486,Z 411.81,A -85,B 0,C 180,E1 2913.558,E2 2913.558} C_VEL
LIN {X 0,Y 267.148,Z 407.91,A -85,B 0,C 180,E1 2910.72,E2 2910.72} C_VEL
LIN {X 0,Y 264.716,Z 403.901,A -85,B 0,C 180,E1 2906.95,E2 2906.95} C_VEL
LIN {X 0,Y 262.238,Z 399.698,A -85,B 0,C 180,E1 2900.067,E2 2900.067} C_VEL
LIN {X 0,Y 262.063,Z 399.47,A -85,B 0,C 180,E1 2893.906,E2 2893.906} C_VEL
LIN {X 0,Y 262.7,Z 400.571,A -85,B 0,C 180,E1 2890.746,E2 2890.746} C_VEL
LIN {X 0,Y 265.495,Z 404.913,A -85,B 0,C 180,E1 2884.534,E2 2884.534} C_VEL
LIN {X 0,Y 268.581,Z 409.801,A -85,B 0,C 180,E1 2880.318,E2 2880.318} C_VEL
LIN {X 0,Y 271.761,Z 414.959,A -85,B 0,C 180,E1 2876.94,E2 2876.94} C_VEL
LIN {X 0,Y 275.917,Z 421.626,A -85,B 0,C 180,E1 2873.339,E2 2873.339} C_VEL
LIN {X 0,Y 281.248,Z 431.015,A -85,B 0,C 180,E1 2869.449,E2 2869.449} C_VEL
LIN {X 0,Y 286.51,Z 440.602,A -85,B 0,C 180,E1 2866.168,E2 2866.168} C_VEL
LIN {X 0,Y 287.459,Z 442.376,A -85,B 0,C 180,E1 2865.615,E2 2865.615} C_VEL
LIN {X 0,Y 287.894,Z 444.382,A -85,B 0,C 180,E1 2865.291,E2 2865.291} C_VEL
LIN {X 0,Y 287.681,Z 448.476,A -85,B 0,C 180,E1 2865.127,E2 2865.127} C_VEL
LIN {X 0,Y 286.449,Z 454.465,A -85,B 0,C 180,E1 2865.296,E2 2865.296} C_VEL
LIN {X 0,Y 284.46,Z 462.723,A -85,B 0,C 180,E1 2865.663,E2 2865.663} C_VEL
LIN {X 0,Y 283.965,Z 466.119,A -85,B 0,C 180,E1 2865.668,E2 2865.668} C_VEL
LIN {X 0,Y 271.444,Z 592.93,A -85,B 0,C 180,E1 2863.039,E2 2863.039} C_VEL
LIN {X 0,Y 267.539,Z 615.1,A -85,B 0,C 180,E1 2862.398,E2 2862.398} C_VEL
LIN {X 0,Y 262.336,Z 635.91,A -85,B 0,C 180,E1 2861.618,E2 2861.618} C_VEL
LIN {X 0,Y 255.569,Z 657.284,A -85,B 0,C 180,E1 2860.528,E2 2860.528} C_VEL
LIN {X 0,Y 248.112,Z 676.805,A -85,B 0,C 180,E1 2859.208,E2 2859.208} C_VEL
LIN {X 0,Y 239.197,Z 696.411,A -85,B 0,C 180,E1 2857.479,E2 2857.479} C_VEL
LIN {X 0,Y 229.768,Z 714.427,A -85,B 0,C 180,E1 2855.427,E2 2855.427} C_VEL
LIN {X 0,Y 218.948,Z 732.701,A -85,B 0,C 180,E1 2852.739,E2 2852.739} C_VEL
LIN {X 0,Y 208.274,Z 748.917,A -85,B 0,C 180,E1 2849.637,E2 2849.637} C_VEL
LIN {X 0,Y 197.083,Z 764.432,A -85,B 0,C 180,E1 2845.78,E2 2845.78} C_VEL
LIN {X 0,Y 186.73,Z 777.733,A -85,B 0,C 180,E1 2841.417,E2 2841.417} C_VEL
LIN {X 0,Y 177.036,Z 789.694,A -85,B 0,C 180,E1 2836.29,E2 2836.29} C_VEL
LIN {X 0,Y 168.409,Z 800.272,A -85,B 0,C 180,E1 2830.321,E2 2830.321} C_VEL
LIN {X 0,Y 161.304,Z 809.389,A -85,B 0,C 180,E1 2823.477,E2 2823.477} C_VEL
LIN {X 0,Y 156.368,Z 816.505,A -85,B 0,C 180,E1 2816.176,E2 2816.176} C_VEL
LIN {X 0,Y 153.575,Z 821.892,A -85,B 0,C 180,E1 2808.599,E2 2808.599} C_VEL
LIN {X 0,Y 152.67,Z 825.509,A -85,B 0,C 180,E1 2801.327,E2 2801.327} C_VEL
LIN {X 0,Y 152.842,Z 827.364,A -85,B 0,C 180,E1 2794.875,E2 2794.875} C_VEL
LIN {X 0,Y 153,Z 827.988,A -85,B 0,C 180,E1 2789.622,E2 2789.622} C_VEL
LIN {X 0,Y 152.754,Z 827.76,A -85,B 0,C 180,E1 2784.362,E2 2784.362} C_VEL
LIN {X 0,Y 152.646,Z 826.329,A -85,B 0,C 180,E1 2777.426,E2 2777.426} C_VEL
LIN {X 0,Y 154.016,Z 823.042,A -85,B 0,C 180,E1 2769.474,E2 2769.474} C_VEL
LIN {X 0,Y 158.093,Z 817.605,A -85,B 0,C 180,E1 2760.853,E2 2760.853} C_VEL
LIN {X 0,Y 164.383,Z 810.929,A -85,B 0,C 180,E1 2753.406,E2 2753.406} C_VEL
LIN {X 0,Y 173.048,Z 802.403,A -85,B 0,C 180,E1 2746.558,E2 2746.558} C_VEL
LIN {X 0,Y 183.308,Z 792.533,A -85,B 0,C 180,E1 2740.692,E2 2740.692} C_VEL
LIN {X 0,Y 195.287,Z 780.796,A -85,B 0,C 180,E1 2735.5,E2 2735.5} C_VEL
LIN {X 0,Y 208.007,Z 767.678,A -85,B 0,C 180,E1 2731.168,E2 2731.168} C_VEL
LIN {X 0,Y 221.077,Z 753.055,A -85,B 0,C 180,E1 2727.566,E2 2727.566} C_VEL
LIN {X 0,Y 233.793,Z 737.467,A -85,B 0,C 180,E1 2724.656,E2 2724.656} C_VEL
LIN {X 0,Y 246.298,Z 720.524,A -85,B 0,C 180,E1 2722.24,E2 2722.24} C_VEL
LIN {X 0,Y 257.989,Z 702.706,A -85,B 0,C 180,E1 2720.295,E2 2720.295} C_VEL
LIN {X 0,Y 268.267,Z 684.729,A -85,B 0,C 180,E1 2718.789,E2 2718.789} C_VEL
LIN {X 0,Y 277.878,Z 665.213,A -85,B 0,C 180,E1 2717.532,E2 2717.532} C_VEL
LIN {X 0,Y 286.474,Z 644.531,A -85,B 0,C 180,E1 2716.533,E2 2716.533} C_VEL
LIN {X 0,Y 293.546,Z 623.558,A -85,B 0,C 180,E1 2715.791,E2 2715.791} C_VEL
LIN {X 0,Y 299.234,Z 601.19,A -85,B 0,C 180,E1 2715.19,E2 2715.19} C_VEL
LIN {X 0,Y 303.101,Z 578.816,A -85,B 0,C 180,E1 2714.711,E2 2714.711} C_VEL
LIN {X 0,Y 317.184,Z 467.819,A -85,B 0,C 180,E1 2712.61,E2 2712.61} C_VEL
LIN {X 0,Y 317.008,Z 467.102,A -85,B 0,C 180,E1 2711.463,E2 2711.463} C_VEL
LIN {X 0,Y 316.989,Z 467.356,A -85,B 0,C 180,E1 2708.893,E2 2708.893} C_VEL
LIN {X 0,Y 316.976,Z 467.906,A -85,B 0,C 180,E1 2708.596,E2 2708.596} C_VEL
LIN {X 0,Y 301.495,Z 584.924,A -85,B 0,C 180,E1 2706.392,E2 2706.392} C_VEL
LIN {X 0,Y 296.959,Z 606.326,A -85,B 0,C 180,E1 2705.805,E2 2705.805} C_VEL
LIN {X 0,Y 291.09,Z 626.66,A -85,B 0,C 180,E1 2705.037,E2 2705.037} C_VEL
LIN {X 0,Y 283.668,Z 646.869,A -85,B 0,C 180,E1 2704.03,E2 2704.03} C_VEL
LIN {X 0,Y 275.303,Z 665.601,A -85,B 0,C 180,E1 2702.824,E2 2702.824} C_VEL
LIN {X 0,Y 265.438,Z 684.097,A -85,B 0,C 180,E1 2701.297,E2 2701.297} C_VEL
LIN {X 0,Y 254.98,Z 700.901,A -85,B 0,C 180,E1 2699.52,E2 2699.52} C_VEL
LIN {X 0,Y 243.248,Z 717.476,A -85,B 0,C 180,E1 2697.278,E2 2697.278} C_VEL
LIN {X 0,Y 231.509,Z 732.131,A -85,B 0,C 180,E1 2694.715,E2 2694.715} C_VEL
LIN {X 0,Y 218.919,Z 746.146,A -85,B 0,C 180,E1 2691.524,E2 2691.524} C_VEL
LIN {X 0,Y 206.631,Z 758.386,A -85,B 0,C 180,E1 2687.82,E2 2687.82} C_VEL
LIN {X 0,Y 194.972,Z 769.029,A -85,B 0,C 180,E1 2683.54,E2 2683.54} C_VEL
LIN {X 0,Y 183.492,Z 778.701,A -85,B 0,C 180,E1 2678.254,E2 2678.254} C_VEL
LIN {X 0,Y 173.751,Z 786.415,A -85,B 0,C 180,E1 2672.406,E2 2672.406} C_VEL
LIN {X 0,Y 165.144,Z 792.852,A -85,B 0,C 180,E1 2665.315,E2 2665.315} C_VEL
LIN {X 0,Y 158.982,Z 797.288,A -85,B 0,C 180,E1 2657.711,E2 2657.711} C_VEL
LIN {X 0,Y 155.283,Z 799.886,A -85,B 0,C 180,E1 2649.989,E2 2649.989} C_VEL
LIN {X 0,Y 153.559,Z 800.906,A -85,B 0,C 180,E1 2642.179,E2 2642.179} C_VEL
LIN {X 0,Y 153.157,Z 800.576,A -85,B 0,C 180,E1 2635.527,E2 2635.527} C_VEL
LIN {X 0,Y 153.529,Z 799.051,A -85,B 0,C 180,E1 2628.613,E2 2628.613} C_VEL
LIN {X 0,Y 155.13,Z 796.044,A -85,B 0,C 180,E1 2621.153,E2 2621.153} C_VEL
LIN {X 0,Y 158.56,Z 791.198,A -85,B 0,C 180,E1 2613.619,E2 2613.619} C_VEL
LIN {X 0,Y 163.605,Z 785.003,A -85,B 0,C 180,E1 2606.851,E2 2606.851} C_VEL
LIN {X 0,Y 170.774,Z 776.71,A -85,B 0,C 180,E1 2600.228,E2 2600.228} C_VEL
LIN {X 0,Y 179.214,Z 766.967,A -85,B 0,C 180,E1 2594.47,E2 2594.47} C_VEL
LIN {X 0,Y 188.521,Z 755.856,A -85,B 0,C 180,E1 2589.514,E2 2589.514} C_VEL
LIN {X 0,Y 198.921,Z 742.53,A -85,B 0,C 180,E1 2585.029,E2 2585.029} C_VEL
LIN {X 0,Y 208.977,Z 728.516,A -85,B 0,C 180,E1 2581.419,E2 2581.419} C_VEL
LIN {X 0,Y 219.336,Z 712.6,A -85,B 0,C 180,E1 2578.233,E2 2578.233} C_VEL
LIN {X 0,Y 229.509,Z 695.007,A -85,B 0,C 180,E1 2575.508,E2 2575.508} C_VEL
LIN {X 0,Y 238.534,Z 677.216,A -85,B 0,C 180,E1 2573.361,E2 2573.361} C_VEL
LIN {X 0,Y 246.842,Z 658.207,A -85,B 0,C 180,E1 2571.558,E2 2571.558} C_VEL
LIN {X 0,Y 254.313,Z 637.668,A -85,B 0,C 180,E1 2570.051,E2 2570.051} C_VEL
LIN {X 0,Y 260.402,Z 616.817,A -85,B 0,C 180,E1 2568.891,E2 2568.891} C_VEL
LIN {X 0,Y 265.168,Z 595.638,A -85,B 0,C 180,E1 2568.018,E2 2568.018} C_VEL
LIN {X 0,Y 268.697,Z 573.268,A -85,B 0,C 180,E1 2567.375,E2 2567.375} C_VEL
LIN {X 0,Y 282.009,Z 445.268,A -85,B 0,C 180,E1 2564.692,E2 2564.692} C_VEL
LIN {X 0,Y 276.733,Z 434.884,A -85,B 0,C 180,E1 2561.044,E2 2561.044} C_VEL
LIN {X 0,Y 272.518,Z 427.205,A -85,B 0,C 180,E1 2557.637,E2 2557.637} C_VEL
LIN {X 0,Y 268.599,Z 420.317,A -85,B 0,C 180,E1 2553.812,E2 2553.812} C_VEL
LIN {X 0,Y 265.7,Z 415.535,A -85,B 0,C 180,E1 2550.279,E2 2550.279} C_VEL
LIN {X 0,Y 263.432,Z 411.665,A -85,B 0,C 180,E1 2546.605,E2 2546.605} C_VEL
LIN {X 0,Y 261.14,Z 407.6,A -85,B 0,C 180,E1 2539.921,E2 2539.921} C_VEL
LIN {X 0,Y 261.022,Z 407.425,A -85,B 0,C 180,E1 2533.737,E2 2533.737} C_VEL
LIN {X 0,Y 261.613,Z 408.541,A -85,B 0,C 180,E1 2530.792,E2 2530.792} C_VEL
LIN {X 0,Y 264.193,Z 412.644,A -85,B 0,C 180,E1 2524.883,E2 2524.883} C_VEL
LIN {X 0,Y 267.103,Z 417.405,A -85,B 0,C 180,E1 2520.749,E2 2520.749} C_VEL
LIN {X 0,Y 270.249,Z 422.678,A -85,B 0,C 180,E1 2517.296,E2 2517.296} C_VEL
LIN {X 0,Y 274.133,Z 429.105,A -85,B 0,C 180,E1 2513.822,E2 2513.822} C_VEL
LIN {X 0,Y 279.355,Z 438.553,A -85,B 0,C 180,E1 2509.898,E2 2509.898} C_VEL
LIN {X 0,Y 284.355,Z 447.965,A -85,B 0,C 180,E1 2506.683,E2 2506.683} C_VEL
LIN {X 0,Y 285.51,Z 450.456,A -85,B 0,C 180,E1 2505.983,E2 2505.983} C_VEL
LIN {X 0,Y 283.965,Z 466.119,A -85,B 0,C 180,E1 2505.668,E2 2505.668} C_VEL
LIN {X 0,Y 282.808,Z 473.796,A -85,B 0,C 180,E1 2505.697,E2 2505.697} C_VEL
LIN {X 0,Y 278.25,Z 494.215,A -85,B 0,C 180,E1 2506.459,E2 2506.459} C_VEL
LIN {X 0,Y 277.286,Z 500.805,A -85,B 0,C 180,E1 2506.469,E2 2506.469} C_VEL
LIN {X 0,Y 267.95,Z 592.784,A -85,B 0,C 180,E1 2504.571,E2 2504.571} C_VEL
LIN {X 0,Y 263.944,Z 615.02,A -85,B 0,C 180,E1 2503.94,E2 2503.94} C_VEL
LIN {X 0,Y 258.53,Z 636.115,A -85,B 0,C 180,E1 2503.166,E2 2503.166} C_VEL
LIN {X 0,Y 251.46,Z 657.782,A -85,B 0,C 180,E1 2502.076,E2 2502.076} C_VEL
LIN {X 0,Y 243.589,Z 677.666,A -85,B 0,C 180,E1 2500.739,E2 2500.739} C_VEL
LIN {X 0,Y 234.479,Z 697.134,A -85,B 0,C 180,E1 2499.035,E2 2499.035} C_VEL
LIN {X 0,Y 224.409,Z 715.656,A -85,B 0,C 180,E1 2496.914,E2 2496.914} C_VEL
LIN {X 0,Y 213.959,Z 732.659,A -85,B 0,C 180,E1 2494.403,E2 2494.403} C_VEL
LIN {X 0,Y 202.894,Z 748.89,A -85,B 0,C 180,E1 2491.297,E2 2491.297} C_VEL
LIN {X 0,Y 191.811,Z 763.728,A -85,B 0,C 180,E1 2487.608,E2 2487.608} C_VEL
LIN {X 0,Y 180.994,Z 777.034,A -85,B 0,C 180,E1 2483.221,E2 2483.221} C_VEL
LIN {X 0,Y 170.806,Z 789.005,A -85,B 0,C 180,E1 2478.018,E2 2478.018} C_VEL
LIN {X 0,Y 161.667,Z 799.598,A -85,B 0,C 180,E1 2471.903,E2 2471.903} C_VEL
LIN {X 0,Y 154.079,Z 808.728,A -85,B 0,C 180,E1 2464.819,E2 2464.819} C_VEL
LIN {X 0,Y 148.757,Z 815.845,A -85,B 0,C 180,E1 2457.193,E2 2457.193} C_VEL
LIN {X 0,Y 145.705,Z 821.219,A -85,B 0,C 180,E1 2449.227,E2 2449.227} C_VEL
LIN {X 0,Y 144.698,Z 824.826,A -85,B 0,C 180,E1 2441.555,E2 2441.555} C_VEL
LIN {X 0,Y 144.879,Z 826.662,A -85,B 0,C 180,E1 2434.746,E2 2434.746} C_VEL
LIN {X 0,Y 145.033,Z 827.253,A -85,B 0,C 180,E1 2429.601,E2 2429.601} C_VEL
LIN {X 0,Y 144.767,Z 827.047,A -85,B 0,C 180,E1 2424.045,E2 2424.045} C_VEL
LIN {X 0,Y 144.695,Z 825.657,A -85,B 0,C 180,E1 2416.815,E2 2416.815} C_VEL
LIN {X 0,Y 146.329,Z 822.405,A -85,B 0,C 180,E1 2408.329,E2 2408.329} C_VEL
LIN {X 0,Y 150.676,Z 817.267,A -85,B 0,C 180,E1 2399.62,E2 2399.62} C_VEL
LIN {X 0,Y 157.768,Z 810.443,A -85,B 0,C 180,E1 2391.601,E2 2391.601} C_VEL
LIN {X 0,Y 167.621,Z 801.537,A -85,B 0,C 180,E1 2384.262,E2 2384.262} C_VEL
LIN {X 0,Y 179.182,Z 791.152,A -85,B 0,C 180,E1 2378.108,E2 2378.108} C_VEL
LIN {X 0,Y 192.609,Z 778.666,A -85,B 0,C 180,E1 2372.753,E2 2372.753} C_VEL
LIN {X 0,Y 206.062,Z 765.348,A -85,B 0,C 180,E1 2368.563,E2 2368.563} C_VEL
LIN {X 0,Y 219.758,Z 750.607,A -85,B 0,C 180,E1 2365.116,E2 2365.116} C_VEL
LIN {X 0,Y 232.985,Z 734.769,A -85,B 0,C 180,E1 2362.354,E2 2362.354} C_VEL
LIN {X 0,Y 245.488,Z 718.112,A -85,B 0,C 180,E1 2360.137,E2 2360.137} C_VEL
LIN {X 0,Y 257.077,Z 700.727,A -85,B 0,C 180,E1 2358.365,E2 2358.365} C_VEL
LIN {X 0,Y 268.039,Z 681.925,A -85,B 0,C 180,E1 2356.895,E2 2356.895} C_VEL
LIN {X 0,Y 277.415,Z 662.992,A -85,B 0,C 180,E1 2355.773,E2 2355.773} C_VEL
LIN {X 0,Y 286.027,Z 642.304,A -85,B 0,C 180,E1 2354.854,E2 2354.854} C_VEL
LIN {X 0,Y 293.058,Z 621.495,A -85,B 0,C 180,E1 2354.176,E2 2354.176} C_VEL
LIN {X 0,Y 298.711,Z 599.497,A -85,B 0,C 180,E1 2353.621,E2 2353.621} C_VEL
LIN {X 0,Y 302.648,Z 576.643,A -85,B 0,C 180,E1 2353.156,E2 2353.156} C_VEL
LIN {X 0,Y 315.907,Z 474.998,A -85,B 0,C 180,E1 2351.272,E2 2351.272} C_VEL
LIN {X 0,Y 315.823,Z 475.175,A -85,B 0,C 180,E1 2349.921,E2 2349.921} C_VEL
LIN {X 0,Y 300.82,Z 585.761,A -85,B 0,C 180,E1 2347.9,E2 2347.9} C_VEL
LIN {X 0,Y 296.198,Z 607.008,A -85,B 0,C 180,E1 2347.34,E2 2347.34} C_VEL
LIN {X 0,Y 290.139,Z 627.43,A -85,B 0,C 180,E1 2346.601,E2 2346.601} C_VEL
LIN {X 0,Y 282.319,Z 648.085,A -85,B 0,C 180,E1 2345.609,E2 2345.609} C_VEL
LIN {X 0,Y 273.796,Z 666.652,A -85,B 0,C 180,E1 2344.457,E2 2344.457} C_VEL
LIN {X 0,Y 263.659,Z 685.082,A -85,B 0,C 180,E1 2342.988,E2 2342.988} C_VEL
LIN {X 0,Y 252.477,Z 702.488,A -85,B 0,C 180,E1 2341.201,E2 2341.201} C_VEL
LIN {X 0,Y 240.501,Z 718.736,A -85,B 0,C 180,E1 2339.049,E2 2339.049} C_VEL
LIN {X 0,Y 227.438,Z 734.337,A -85,B 0,C 180,E1 2336.346,E2 2336.346} C_VEL
LIN {X 0,Y 214.483,Z 748.067,A -85,B 0,C 180,E1 2333.209,E2 2333.209} C_VEL
LIN {X 0,Y 201.01,Z 760.828,A -85,B 0,C 180,E1 2329.293,E2 2329.293} C_VEL
LIN {X 0,Y 188.546,Z 771.428,A -85,B 0,C 180,E1 2324.838,E2 2324.838} C_VEL
LIN {X 0,Y 176.659,Z 780.727,A -85,B 0,C 180,E1 2319.46,E2 2319.46} C_VEL
LIN {X 0,Y 165.979,Z 788.487,A -85,B 0,C 180,E1 2313.076,E2 2313.076} C_VEL
LIN {X 0,Y 157.485,Z 794.319,A -85,B 0,C 180,E1 2306.038,E2 2306.038} C_VEL
LIN {X 0,Y 151.068,Z 798.562,A -85,B 0,C 180,E1 2298.055,E2 2298.055} C_VEL
LIN {X 0,Y 147.177,Z 800.947,A -85,B 0,C 180,E1 2289.692,E2 2289.692} C_VEL
LIN {X 0,Y 145.556,Z 801.651,A -85,B 0,C 180,E1 2281.938,E2 2281.938} C_VEL
LIN {X 0,Y 145.194,Z 801.184,A -85,B 0,C 180,E1 2274.642,E2 2274.642} C_VEL
LIN {X 0,Y 145.695,Z 799.451,A -85,B 0,C 180,E1 2267.477,E2 2267.477} C_VEL
LIN {X 0,Y 147.721,Z 796.053,A -85,B 0,C 180,E1 2259.353,E2 2259.353} C_VEL
LIN {X 0,Y 151.474,Z 791.314,A -85,B 0,C 180,E1 2251.895,E2 2251.895} C_VEL
LIN {X 0,Y 157.413,Z 784.55,A -85,B 0,C 180,E1 2244.537,E2 2244.537} C_VEL
LIN {X 0,Y 164.873,Z 776.391,A -85,B 0,C 180,E1 2238.105,E2 2238.105} C_VEL
LIN {X 0,Y 173.94,Z 766.402,A -85,B 0,C 180,E1 2232.266,E2 2232.266} C_VEL
LIN {X 0,Y 183.829,Z 755.031,A -85,B 0,C 180,E1 2227.287,E2 2227.287} C_VEL
LIN {X 0,Y 194.171,Z 742.313,A -85,B 0,C 180,E1 2223.058,E2 2223.058} C_VEL
LIN {X 0,Y 204.656,Z 728.136,A -85,B 0,C 180,E1 2219.467,E2 2219.467} C_VEL
LIN {X 0,Y 215.055,Z 712.581,A -85,B 0,C 180,E1 2216.412,E2 2216.412} C_VEL
LIN {X 0,Y 225.192,Z 695.526,A -85,B 0,C 180,E1 2213.81,E2 2213.81} C_VEL
LIN {X 0,Y 234.561,Z 677.518,A -85,B 0,C 180,E1 2211.672,E2 2211.672} C_VEL
LIN {X 0,Y 243,Z 658.663,A -85,B 0,C 180,E1 2209.917,E2 2209.917} C_VEL
LIN {X 0,Y 250.395,Z 638.826,A -85,B 0,C 180,E1 2208.486,E2 2208.486} C_VEL
LIN {X 0,Y 256.494,Z 618.631,A -85,B 0,C 180,E1 2207.37,E2 2207.37} C_VEL
LIN {X 0,Y 261.566,Z 596.958,A -85,B 0,C 180,E1 2206.479,E2 2206.479} C_VEL
LIN {X 0,Y 265.301,Z 574.113,A -85,B 0,C 180,E1 2205.827,E2 2205.827} C_VEL
LIN {X 0,Y 278.576,Z 449.789,A -85,B 0,C 180,E1 2203.274,E2 2203.274} C_VEL
LIN {X 0,Y 273.095,Z 438.964,A -85,B 0,C 180,E1 2199.149,E2 2199.149} C_VEL
LIN {X 0,Y 269.116,Z 431.61,A -85,B 0,C 180,E1 2195.55,E2 2195.55} C_VEL
LIN {X 0,Y 266.274,Z 426.692,A -85,B 0,C 180,E1 2192.475,E2 2192.475} C_VEL
LIN {X 0,Y 264.268,Z 423.158,A -85,B 0,C 180,E1 2189.834,E2 2189.834} C_VEL
LIN {X 0,Y 262.158,Z 419.429,A -85,B 0,C 180,E1 2186.256,E2 2186.256} C_VEL
LIN {X 0,Y 260.044,Z 415.503,A -85,B 0,C 180,E1 2179.775,E2 2179.775} C_VEL
LIN {X 0,Y 259.977,Z 415.388,A -85,B 0,C 180,E1 2173.566,E2 2173.566} C_VEL
LIN {X 0,Y 260.542,Z 416.563,A -85,B 0,C 180,E1 2170.773,E2 2170.773} C_VEL
LIN {X 0,Y 262.898,Z 420.375,A -85,B 0,C 180,E1 2165.235,E2 2165.235} C_VEL
LIN {X 0,Y 265.718,Z 425.171,A -85,B 0,C 180,E1 2161.076,E2 2161.076} C_VEL
LIN {X 0,Y 268.54,Z 430.026,A -85,B 0,C 180,E1 2157.864,E2 2157.864} C_VEL
LIN {X 0,Y 272.301,Z 436.459,A -85,B 0,C 180,E1 2154.365,E2 2154.365} C_VEL
LIN {X 0,Y 277.54,Z 446.211,A -85,B 0,C 180,E1 2150.302,E2 2150.302} C_VEL
LIN {X 0,Y 281.922,Z 454.764,A -85,B 0,C 180,E1 2147.384,E2 2147.384} C_VEL
LIN {X 0,Y 277.286,Z 500.805,A -85,B 0,C 180,E1 2146.469,E2 2146.469} C_VEL
LIN {X 0,Y 276.12,Z 508.481,A -85,B 0,C 180,E1 2146.503,E2 2146.503} C_VEL
LIN {X 0,Y 271.608,Z 528.898,A -85,B 0,C 180,E1 2147.294,E2 2147.294} C_VEL
LIN {X 0,Y 270.642,Z 535.488,A -85,B 0,C 180,E1 2147.312,E2 2147.312} C_VEL
LIN {X 0,Y 264.539,Z 592.839,A -85,B 0,C 180,E1 2146.129,E2 2146.129} C_VEL
LIN {X 0,Y 260.422,Z 615.113,A -85,B 0,C 180,E1 2145.51,E2 2145.51} C_VEL
LIN {X 0,Y 254.917,Z 636.058,A -85,B 0,C 180,E1 2144.76,E2 2144.76} C_VEL
LIN {X 0,Y 247.883,Z 657.197,A -85,B 0,C 180,E1 2143.728,E2 2143.728} C_VEL
LIN {X 0,Y 240.105,Z 676.559,A -85,B 0,C 180,E1 2142.47,E2 2142.47} C_VEL
LIN {X 0,Y 230.777,Z 696.114,A -85,B 0,C 180,E1 2140.812,E2 2140.812} C_VEL
LIN {X 0,Y 220.863,Z 714.024,A -85,B 0,C 180,E1 2138.83,E2 2138.83} C_VEL
LIN {X 0,Y 209.682,Z 731.814,A -85,B 0,C 180,E1 2136.274,E2 2136.274} C_VEL
LIN {X 0,Y 198.445,Z 747.823,A -85,B 0,C 180,E1 2133.265,E2 2133.265} C_VEL
LIN {X 0,Y 186.742,Z 762.943,A -85,B 0,C 180,E1 2129.538,E2 2129.538} C_VEL
LIN {X 0,Y 175.449,Z 776.297,A -85,B 0,C 180,E1 2125.141,E2 2125.141} C_VEL
LIN {X 0,Y 164.743,Z 788.306,A -85,B 0,C 180,E1 2119.875,E2 2119.875} C_VEL
LIN {X 0,Y 155.059,Z 798.912,A -85,B 0,C 180,E1 2113.621,E2 2113.621} C_VEL
LIN {X 0,Y 146.946,Z 808.042,A -85,B 0,C 180,E1 2106.291,E2 2106.291} C_VEL
LIN {X 0,Y 141.195,Z 815.163,A -85,B 0,C 180,E1 2098.319,E2 2098.319} C_VEL
LIN {X 0,Y 137.851,Z 820.536,A -85,B 0,C 180,E1 2089.927,E2 2089.927} C_VEL
LIN {X 0,Y 136.729,Z 824.139,A -85,B 0,C 180,E1 2081.811,E2 2081.811} C_VEL
LIN {X 0,Y 136.917,Z 825.956,A -85,B 0,C 180,E1 2074.603,E2 2074.603} C_VEL
LIN {X 0,Y 137.054,Z 826.525,A -85,B 0,C 180,E1 2069.16,E2 2069.16} C_VEL
LIN {X 0,Y 136.769,Z 826.335,A -85,B 0,C 180,E1 2063.7,E2 2063.7} C_VEL
LIN {X 0,Y 136.732,Z 825.064,A -85,B 0,C 180,E1 2056.463,E2 2056.463} C_VEL
LIN {X 0,Y 138.538,Z 821.969,A -85,B 0,C 180,E1 2047.495,E2 2047.495} C_VEL
LIN {X 0,Y 143.244,Z 817.037,A -85,B 0,C 180,E1 2038.388,E2 2038.388} C_VEL
LIN {X 0,Y 151.319,Z 809.955,A -85,B 0,C 180,E1 2029.639,E2 2029.639} C_VEL
LIN {X 0,Y 161.348,Z 801.593,A -85,B 0,C 180,E1 2022.482,E2 2022.482} C_VEL
LIN {X 0,Y 173.547,Z 791.418,A -85,B 0,C 180,E1 2016.232,E2 2016.232} C_VEL
LIN {X 0,Y 186.859,Z 779.862,A -85,B 0,C 180,E1 2011.109,E2 2011.109} C_VEL
LIN {X 0,Y 200.743,Z 766.899,A -85,B 0,C 180,E1 2006.925,E2 2006.925} C_VEL
LIN {X 0,Y 214.007,Z 753.334,A -85,B 0,C 180,E1 2003.685,E2 2003.685} C_VEL
LIN {X 0,Y 228.583,Z 736.929,A -85,B 0,C 180,E1 2000.753,E2 2000.753} C_VEL
LIN {X 0,Y 241.543,Z 720.574,A -85,B 0,C 180,E1 1998.564,E2 1998.564} C_VEL
LIN {X 0,Y 253.346,Z 703.767,A -85,B 0,C 180,E1 1996.847,E2 1996.847} C_VEL
LIN {X 0,Y 264.497,Z 685.525,A -85,B 0,C 180,E1 1995.423,E2 1995.423} C_VEL
LIN {X 0,Y 274.931,Z 665.748,A -85,B 0,C 180,E1 1994.251,E2 1994.251} C_VEL
LIN {X 0,Y 283.668,Z 646.052,A -85,B 0,C 180,E1 1993.38,E2 1993.38} C_VEL
LIN {X 0,Y 291.1,Z 625.277,A -85,B 0,C 180,E1 1992.71,E2 1992.71} C_VEL
LIN {X 0,Y 297.027,Z 603.908,A -85,B 0,C 180,E1 1992.179,E2 1992.179} C_VEL
LIN {X 0,Y 301.5,Z 581.083,A -85,B 0,C 180,E1 1991.719,E2 1991.719} C_VEL
LIN {X 0,Y 309.801,Z 519.541,A -85,B 0,C 180,E1 1990.617,E2 1990.617} C_VEL
LIN {X 0,Y 300.466,Z 586.409,A -85,B 0,C 180,E1 1989.419,E2 1989.419} C_VEL
LIN {X 0,Y 295.742,Z 607.604,A -85,B 0,C 180,E1 1988.885,E2 1988.885} C_VEL
LIN {X 0,Y 289.608,Z 627.813,A -85,B 0,C 180,E1 1988.19,E2 1988.19} C_VEL
LIN {X 0,Y 281.724,Z 648.334,A -85,B 0,C 180,E1 1987.256,E2 1987.256} C_VEL
LIN {X 0,Y 273.048,Z 666.84,A -85,B 0,C 180,E1 1986.167,E2 1986.167} C_VEL
LIN {X 0,Y 262.364,Z 685.792,A -85,B 0,C 180,E1 1984.728,E2 1984.728} C_VEL
LIN {X 0,Y 251.337,Z 702.531,A -85,B 0,C 180,E1 1983.09,E2 1983.09} C_VEL
LIN {X 0,Y 238.598,Z 719.347,A -85,B 0,C 180,E1 1980.962,E2 1980.962} C_VEL
LIN {X 0,Y 225.705,Z 734.313,A -85,B 0,C 180,E1 1978.479,E2 1978.479} C_VEL
LIN {X 0,Y 212.047,Z 748.329,A -85,B 0,C 180,E1 1975.405,E2 1975.405} C_VEL
LIN {X 0,Y 198.525,Z 760.6,A -85,B 0,C 180,E1 1971.77,E2 1971.77} C_VEL
LIN {X 0,Y 185.42,Z 771.328,A -85,B 0,C 180,E1 1967.44,E2 1967.44} C_VEL
LIN {X 0,Y 172.423,Z 780.975,A -85,B 0,C 180,E1 1962.001,E2 1962.001} C_VEL
LIN {X 0,Y 161.168,Z 788.67,A -85,B 0,C 180,E1 1955.786,E2 1955.786} C_VEL
LIN {X 0,Y 151.474,Z 794.83,A -85,B 0,C 180,E1 1948.383,E2 1948.383} C_VEL
LIN {X 0,Y 144.338,Z 799.067,A -85,B 0,C 180,E1 1940.262,E2 1940.262} C_VEL
LIN {X 0,Y 139.838,Z 801.526,A -85,B 0,C 180,E1 1931.684,E2 1931.684} C_VEL
LIN {X 0,Y 137.715,Z 802.392,A -85,B 0,C 180,E1 1922.997,E2 1922.997} C_VEL
LIN {X 0,Y 137.218,Z 801.973,A -85,B 0,C 180,E1 1915.466,E2 1915.466} C_VEL
LIN {X 0,Y 137.676,Z 800.305,A -85,B 0,C 180,E1 1907.764,E2 1907.764} C_VEL
LIN {X 0,Y 139.632,Z 797.166,A -85,B 0,C 180,E1 1899.484,E2 1899.484} C_VEL
LIN {X 0,Y 143.723,Z 792.248,A -85,B 0,C 180,E1 1891.2,E2 1891.2} C_VEL
LIN {X 0,Y 149.976,Z 785.551,A -85,B 0,C 180,E1 1883.496,E2 1883.496} C_VEL
LIN {X 0,Y 157.815,Z 777.477,A -85,B 0,C 180,E1 1876.82,E2 1876.82} C_VEL
LIN {X 0,Y 167.304,Z 767.577,A -85,B 0,C 180,E1 1870.814,E2 1870.814} C_VEL
LIN {X 0,Y 177.609,Z 756.304,A -85,B 0,C 180,E1 1865.739,E2 1865.739} C_VEL
LIN {X 0,Y 188.994,Z 742.849,A -85,B 0,C 180,E1 1861.225,E2 1861.225} C_VEL
LIN {X 0,Y 200.326,Z 728.038,A -85,B 0,C 180,E1 1857.506,E2 1857.506} C_VEL
LIN {X 0,Y 210.992,Z 712.487,A -85,B 0,C 180,E1 1854.518,E2 1854.518} C_VEL
LIN {X 0,Y 221.296,Z 695.555,A -85,B 0,C 180,E1 1851.993,E2 1851.993} C_VEL
LIN {X 0,Y 231.088,Z 677.105,A -85,B 0,C 180,E1 1849.862,E2 1849.862} C_VEL
LIN {X 0,Y 239.355,Z 659.024,A -85,B 0,C 180,E1 1848.223,E2 1848.223} C_VEL
LIN {X 0,Y 246.931,Z 639.162,A -85,B 0,C 180,E1 1846.823,E2 1846.823} C_VEL
LIN {X 0,Y 253.171,Z 618.926,A -85,B 0,C 180,E1 1845.734,E2 1845.734} C_VEL
LIN {X 0,Y 258.331,Z 597.323,A -85,B 0,C 180,E1 1844.868,E2 1844.868} C_VEL
LIN {X 0,Y 262.148,Z 574.46,A -85,B 0,C 180,E1 1844.232,E2 1844.232} C_VEL
LIN {X 0,Y 275.235,Z 454.52,A -85,B 0,C 180,E1 1841.796,E2 1841.796} C_VEL
LIN {X 0,Y 270.589,Z 444.995,A -85,B 0,C 180,E1 1838.033,E2 1838.033} C_VEL
LIN {X 0,Y 266.94,Z 438.207,A -85,B 0,C 180,E1 1834.514,E2 1834.514} C_VEL
LIN {X 0,Y 264.528,Z 433.811,A -85,B 0,C 180,E1 1831.692,E2 1831.692} C_VEL
LIN {X 0,Y 262.853,Z 430.78,A -85,B 0,C 180,E1 1829.384,E2 1829.384} C_VEL
LIN {X 0,Y 260.895,Z 427.193,A -85,B 0,C 180,E1 1825.904,E2 1825.904} C_VEL
LIN {X 0,Y 258.943,Z 423.398,A -85,B 0,C 180,E1 1819.591,E2 1819.591} C_VEL
LIN {X 0,Y 258.935,Z 423.354,A -85,B 0,C 180,E1 1813.394,E2 1813.394} C_VEL
LIN {X 0,Y 259.498,Z 424.656,A -85,B 0,C 180,E1 1810.656,E2 1810.656} C_VEL
LIN {X 0,Y 261.668,Z 428.24,A -85,B 0,C 180,E1 1805.48,E2 1805.48} C_VEL
LIN {X 0,Y 264.261,Z 432.772,A -85,B 0,C 180,E1 1801.516,E2 1801.516} C_VEL
LIN {X 0,Y 267.141,Z 437.908,A -85,B 0,C 180,E1 1798.133,E2 1798.133} C_VEL
LIN {X 0,Y 270.62,Z 444.057,A -85,B 0,C 180,E1 1794.805,E2 1794.805} C_VEL
LIN {X 0,Y 275.951,Z 454.256,A -85,B 0,C 180,E1 1790.562,E2 1790.562} C_VEL
LIN {X 0,Y 278.443,Z 459.506,A -85,B 0,C 180,E1 1788.811,E2 1788.811} C_VEL
LIN {X 0,Y 270.642,Z 535.488,A -85,B 0,C 180,E1 1787.312,E2 1787.312} C_VEL
LIN {X 0,Y 269.462,Z 543.164,A -85,B 0,C 180,E1 1787.358,E2 1787.358} C_VEL
LIN {X 0,Y 264.96,Z 563.563,A -85,B 0,C 180,E1 1788.195,E2 1788.195} C_VEL
LIN {X 0,Y 263.999,Z 570.15,A -85,B 0,C 180,E1 1788.21,E2 1788.21} C_VEL
LIN {X 0,Y 260.572,Z 597.411,A -85,B 0,C 180,E1 1787.612,E2 1787.612} C_VEL
LIN {X 0,Y 256.141,Z 619.12,A -85,B 0,C 180,E1 1787,E2 1787} C_VEL
LIN {X 0,Y 250.152,Z 640.474,A -85,B 0,C 180,E1 1786.22,E2 1786.22} C_VEL
LIN {X 0,Y 242.563,Z 661.68,A -85,B 0,C 180,E1 1785.143,E2 1785.143} C_VEL
LIN {X 0,Y 234.219,Z 680.98,A -85,B 0,C 180,E1 1783.832,E2 1783.832} C_VEL
LIN {X 0,Y 223.881,Z 701.278,A -85,B 0,C 180,E1 1782.027,E2 1782.027} C_VEL
LIN {X 0,Y 213.399,Z 719.114,A -85,B 0,C 180,E1 1779.945,E2 1779.945} C_VEL
LIN {X 0,Y 202.037,Z 736.144,A -85,B 0,C 180,E1 1777.354,E2 1777.354} C_VEL
LIN {X 0,Y 190.021,Z 752.134,A -85,B 0,C 180,E1 1774.12,E2 1774.12} C_VEL
LIN {X 0,Y 178.321,Z 766.256,A -85,B 0,C 180,E1 1770.346,E2 1770.346} C_VEL
LIN {X 0,Y 166.558,Z 779.417,A -85,B 0,C 180,E1 1765.644,E2 1765.644} C_VEL
LIN {X 0,Y 155.431,Z 791.199,A -85,B 0,C 180,E1 1759.945,E2 1759.945} C_VEL
LIN {X 0,Y 145.304,Z 801.63,A -85,B 0,C 180,E1 1752.934,E2 1752.934} C_VEL
LIN {X 0,Y 137.444,Z 810.006,A -85,B 0,C 180,E1 1745.073,E2 1745.073} C_VEL
LIN {X 0,Y 131.908,Z 816.819,A -85,B 0,C 180,E1 1736.075,E2 1736.075} C_VEL
LIN {X 0,Y 129.245,Z 821.563,A -85,B 0,C 180,E1 1727.091,E2 1727.091} C_VEL
LIN {X 0,Y 128.746,Z 824.295,A -85,B 0,C 180,E1 1718.931,E2 1718.931} C_VEL
LIN {X 0,Y 129.038,Z 825.503,A -85,B 0,C 180,E1 1712.66,E2 1712.66} C_VEL
LIN {X 0,Y 129.032,Z 825.808,A -85,B 0,C 180,E1 1707.775,E2 1707.775} C_VEL
LIN {X 0,Y 128.68,Z 825.429,A -85,B 0,C 180,E1 1701.506,E2 1701.506} C_VEL
LIN {X 0,Y 129.224,Z 823.564,A -85,B 0,C 180,E1 1692.432,E2 1692.432} C_VEL
LIN {X 0,Y 132.166,Z 820.099,A -85,B 0,C 180,E1 1683.219,E2 1683.219} C_VEL
LIN {X 0,Y 138.188,Z 814.822,A -85,B 0,C 180,E1 1674.116,E2 1674.116} C_VEL
LIN {X 0,Y 147.408,Z 807.66,A -85,B 0,C 180,E1 1665.677,E2 1665.677} C_VEL
LIN {X 0,Y 158.987,Z 798.883,A -85,B 0,C 180,E1 1658.51,E2 1658.51} C_VEL
LIN {X 0,Y 172.126,Z 788.517,A -85,B 0,C 180,E1 1652.612,E2 1652.612} C_VEL
LIN {X 0,Y 186.418,Z 776.547,A -85,B 0,C 180,E1 1647.745,E2 1647.745} C_VEL
LIN {X 0,Y 201.126,Z 763.18,A -85,B 0,C 180,E1 1643.828,E2 1643.828} C_VEL
LIN {X 0,Y 215.021,Z 749.353,A -85,B 0,C 180,E1 1640.821,E2 1640.821} C_VEL
LIN {X 0,Y 229.493,Z 733.174,A -85,B 0,C 180,E1 1638.228,E2 1638.228} C_VEL
LIN {X 0,Y 242.651,Z 716.609,A -85,B 0,C 180,E1 1636.235,E2 1636.235} C_VEL
LIN {X 0,Y 255.224,Z 698.667,A -85,B 0,C 180,E1 1634.609,E2 1634.609} C_VEL
LIN {X 0,Y 266.643,Z 679.874,A -85,B 0,C 180,E1 1633.32,E2 1633.32} C_VEL
LIN {X 0,Y 276.849,Z 659.944,A -85,B 0,C 180,E1 1632.305,E2 1632.305} C_VEL
LIN {X 0,Y 285.258,Z 640.252,A -85,B 0,C 180,E1 1631.564,E2 1631.564} C_VEL
LIN {X 0,Y 292.535,Z 619.128,A -85,B 0,C 180,E1 1630.975,E2 1630.975} C_VEL
LIN {X 0,Y 297.023,Z 602.479,A -85,B 0,C 180,E1 1630.588,E2 1630.588} C_VEL
LIN {X 0,Y 291.379,Z 622.57,A -85,B 0,C 180,E1 1629.984,E2 1629.984} C_VEL
LIN {X 0,Y 284.125,Z 642.243,A -85,B 0,C 180,E1 1629.204,E2 1629.204} C_VEL
LIN {X 0,Y 275.287,Z 661.677,A -85,B 0,C 180,E1 1628.206,E2 1628.206} C_VEL
LIN {X 0,Y 264.897,Z 680.74,A -85,B 0,C 180,E1 1626.939,E2 1626.939} C_VEL
LIN {X 0,Y 254.141,Z 697.592,A -85,B 0,C 180,E1 1625.499,E2 1625.499} C_VEL
LIN {X 0,Y 241.132,Z 715.029,A -85,B 0,C 180,E1 1623.568,E2 1623.568} C_VEL
LIN {X 0,Y 228.038,Z 730.283,A -85,B 0,C 180,E1 1621.337,E2 1621.337} C_VEL
LIN {X 0,Y 214.045,Z 744.663,A -85,B 0,C 180,E1 1618.561,E2 1618.561} C_VEL
LIN {X 0,Y 200.158,Z 757.316,A -85,B 0,C 180,E1 1615.281,E2 1615.281} C_VEL
LIN {X 0,Y 186.148,Z 768.728,A -85,B 0,C 180,E1 1611.251,E2 1611.251} C_VEL
LIN {X 0,Y 172.003,Z 778.96,A -85,B 0,C 180,E1 1606.127,E2 1606.127} C_VEL
LIN {X 0,Y 159.433,Z 787.169,A -85,B 0,C 180,E1 1600.178,E2 1600.178} C_VEL
LIN {X 0,Y 148.221,Z 793.875,A -85,B 0,C 180,E1 1592.936,E2 1592.936} C_VEL
LIN {X 0,Y 139.531,Z 798.669,A -85,B 0,C 180,E1 1584.783,E2 1584.783} C_VEL
LIN {X 0,Y 133.589,Z 801.726,A -85,B 0,C 180,E1 1575.894,E2 1575.894} C_VEL
LIN {X 0,Y 130.386,Z 803.061,A -85,B 0,C 180,E1 1566.742,E2 1566.742} C_VEL
LIN {X 0,Y 129.31,Z 802.913,A -85,B 0,C 180,E1 1558.148,E2 1558.148} C_VEL
LIN {X 0,Y 129.433,Z 801.748,A -85,B 0,C 180,E1 1550.347,E2 1550.347} C_VEL
LIN {X 0,Y 130.84,Z 799.138,A -85,B 0,C 180,E1 1541.912,E2 1541.912} C_VEL
LIN {X 0,Y 134.453,Z 794.765,A -85,B 0,C 180,E1 1532.988,E2 1532.988} C_VEL
LIN {X 0,Y 140.031,Z 789.091,A -85,B 0,C 180,E1 1525.089,E2 1525.089} C_VEL
LIN {X 0,Y 148.045,Z 781.28,A -85,B 0,C 180,E1 1517.523,E2 1517.523} C_VEL
LIN {X 0,Y 157.471,Z 772.02,A -85,B 0,C 180,E1 1511.11,E2 1511.11} C_VEL
LIN {X 0,Y 167.807,Z 761.438,A -85,B 0,C 180,E1 1505.728,E2 1505.728} C_VEL
LIN {X 0,Y 178.62,Z 749.611,A -85,B 0,C 180,E1 1501.227,E2 1501.227} C_VEL
LIN {X 0,Y 190.288,Z 735.652,A -85,B 0,C 180,E1 1497.238,E2 1497.238} C_VEL
LIN {X 0,Y 201.918,Z 720.077,A -85,B 0,C 180,E1 1493.899,E2 1493.899} C_VEL
LIN {X 0,Y 212.511,Z 704.065,A -85,B 0,C 180,E1 1491.266,E2 1491.266} C_VEL
LIN {X 0,Y 222.669,Z 686.616,A -85,B 0,C 180,E1 1489.04,E2 1489.04} C_VEL
LIN {X 0,Y 231.867,Z 668.363,A -85,B 0,C 180,E1 1487.225,E2 1487.225} C_VEL
LIN {X 0,Y 240.243,Z 648.748,A -85,B 0,C 180,E1 1485.708,E2 1485.708} C_VEL
LIN {X 0,Y 247.386,Z 628.251,A -85,B 0,C 180,E1 1484.495,E2 1484.495} C_VEL
LIN {X 0,Y 253.107,Z 607.392,A -85,B 0,C 180,E1 1483.57,E2 1483.57} C_VEL
LIN {X 0,Y 257.5,Z 585.814,A -85,B 0,C 180,E1 1482.874,E2 1482.874} C_VEL
LIN {X 0,Y 261.206,Z 557.337,A -85,B 0,C 180,E1 1482.245,E2 1482.245} C_VEL
LIN {X 0,Y 272.031,Z 459.247,A -85,B 0,C 180,E1 1480.305,E2 1480.305} C_VEL
LIN {X 0,Y 267.657,Z 450.127,A -85,B 0,C 180,E1 1476.436,E2 1476.436} C_VEL
LIN {X 0,Y 263.964,Z 442.964,A -85,B 0,C 180,E1 1472.408,E2 1472.408} C_VEL
LIN {X 0,Y 261.527,Z 438.516,A -85,B 0,C 180,E1 1469.045,E2 1469.045} C_VEL
LIN {X 0,Y 259.641,Z 434.955,A -85,B 0,C 180,E1 1465.548,E2 1465.548} C_VEL
LIN {X 0,Y 257.856,Z 431.31,A -85,B 0,C 180,E1 1459.477,E2 1459.477} C_VEL
LIN {X 0,Y 257.862,Z 431.278,A -85,B 0,C 180,E1 1453.451,E2 1453.451} C_VEL
LIN {X 0,Y 258.418,Z 432.655,A -85,B 0,C 180,E1 1450.669,E2 1450.669} C_VEL
LIN {X 0,Y 260.385,Z 435.957,A -85,B 0,C 180,E1 1445.85,E2 1445.85} C_VEL
LIN {X 0,Y 262.897,Z 440.536,A -85,B 0,C 180,E1 1441.851,E2 1441.851} C_VEL
LIN {X 0,Y 265.578,Z 445.457,A -85,B 0,C 180,E1 1438.596,E2 1438.596} C_VEL
LIN {X 0,Y 268.897,Z 451.53,A -85,B 0,C 180,E1 1435.306,E2 1435.306} C_VEL
LIN {X 0,Y 273.882,Z 461.42,A -85,B 0,C 180,E1 1431.179,E2 1431.179} C_VEL
LIN {X 0,Y 275.092,Z 464.111,A -85,B 0,C 180,E1 1430.27,E2 1430.27} C_VEL
LIN {X 0,Y 263.999,Z 570.15,A -85,B 0,C 180,E1 1428.21,E2 1428.21} C_VEL
LIN {X 0,Y 262.825,Z 577.828,A -85,B 0,C 180,E1 1428.255,E2 1428.255} C_VEL
LIN {X 0,Y 257.733,Z 598.123,A -85,B 0,C 180,E1 1429.085,E2 1429.085} C_VEL
LIN {X 0,Y 256.205,Z 604.606,A -85,B 0,C 180,E1 1429.064,E2 1429.064} C_VEL
LIN {X 0,Y 250.945,Z 626.762,A -85,B 0,C 180,E1 1428.408,E2 1428.408} C_VEL
LIN {X 0,Y 244.419,Z 647.431,A -85,B 0,C 180,E1 1427.584,E2 1427.584} C_VEL
LIN {X 0,Y 236.503,Z 667.801,A -85,B 0,C 180,E1 1426.486,E2 1426.486} C_VEL
LIN {X 0,Y 227.593,Z 687.037,A -85,B 0,C 180,E1 1425.115,E2 1425.115} C_VEL
LIN {X 0,Y 217.1,Z 706.332,A -85,B 0,C 180,E1 1423.313,E2 1423.313} C_VEL
LIN {X 0,Y 206.021,Z 723.874,A -85,B 0,C 180,E1 1421.139,E2 1421.139} C_VEL
LIN {X 0,Y 194.061,Z 740.591,A -85,B 0,C 180,E1 1418.423,E2 1418.423} C_VEL
LIN {X 0,Y 181.84,Z 755.908,A -85,B 0,C 180,E1 1415.121,E2 1415.121} C_VEL
LIN {X 0,Y 169.511,Z 769.964,A -85,B 0,C 180,E1 1411.072,E2 1411.072} C_VEL
LIN {X 0,Y 157.079,Z 782.948,A -85,B 0,C 180,E1 1405.931,E2 1405.931} C_VEL
LIN {X 0,Y 145.91,Z 793.962,A -85,B 0,C 180,E1 1399.895,E2 1399.895} C_VEL
LIN {X 0,Y 136.001,Z 803.595,A -85,B 0,C 180,E1 1392.554,E2 1392.554} C_VEL
LIN {X 0,Y 128.56,Z 811.219,A -85,B 0,C 180,E1 1384.467,E2 1384.467} C_VEL
LIN {X 0,Y 123.498,Z 817.207,A -85,B 0,C 180,E1 1375.405,E2 1375.405} C_VEL
LIN {X 0,Y 121.071,Z 821.549,A -85,B 0,C 180,E1 1365.809,E2 1365.809} C_VEL
LIN {X 0,Y 120.812,Z 823.943,A -85,B 0,C 180,E1 1357.604,E2 1357.604} C_VEL
LIN {X 0,Y 121.124,Z 824.968,A -85,B 0,C 180,E1 1350.941,E2 1350.941} C_VEL
LIN {X 0,Y 120.883,Z 825.075,A -85,B 0,C 180,E1 1344.775,E2 1344.775} C_VEL
LIN {X 0,Y 120.783,Z 823.99,A -85,B 0,C 180,E1 1336.105,E2 1336.105} C_VEL
LIN {X 0,Y 122.88,Z 821.309,A -85,B 0,C 180,E1 1325.988,E2 1325.988} C_VEL
LIN {X 0,Y 128.332,Z 816.685,A -85,B 0,C 180,E1 1315.872,E2 1315.872} C_VEL
LIN {X 0,Y 137.101,Z 810.343,A -85,B 0,C 180,E1 1306.718,E2 1306.718} C_VEL
LIN {X 0,Y 148.801,Z 802.179,A -85,B 0,C 180,E1 1298.784,E2 1298.784} C_VEL
LIN {X 0,Y 162.213,Z 792.562,A -85,B 0,C 180,E1 1292.381,E2 1292.381} C_VEL
LIN {X 0,Y 176.607,Z 781.495,A -85,B 0,C 180,E1 1287.264,E2 1287.264} C_VEL
LIN {X 0,Y 192.242,Z 768.442,A -85,B 0,C 180,E1 1282.982,E2 1282.982} C_VEL
LIN {X 0,Y 207.999,Z 753.866,A -85,B 0,C 180,E1 1279.573,E2 1279.573} C_VEL
LIN {X 0,Y 222.258,Z 739.236,A -85,B 0,C 180,E1 1277.061,E2 1277.061} C_VEL
LIN {X 0,Y 236.568,Z 722.55,A -85,B 0,C 180,E1 1274.942,E2 1274.942} C_VEL
LIN {X 0,Y 249.173,Z 705.859,A -85,B 0,C 180,E1 1273.354,E2 1273.354} C_VEL
LIN {X 0,Y 261.683,Z 686.887,A -85,B 0,C 180,E1 1271.993,E2 1271.993} C_VEL
LIN {X 0,Y 271.977,Z 668.74,A -85,B 0,C 180,E1 1271.012,E2 1271.012} C_VEL
LIN {X 0,Y 279.463,Z 653.18,A -85,B 0,C 180,E1 1270.359,E2 1270.359} C_VEL
LIN {X 0,Y 269.496,Z 672.646,A -85,B 0,C 180,E1 1269.279,E2 1269.279} C_VEL
LIN {X 0,Y 258.475,Z 690.705,A -85,B 0,C 180,E1 1267.982,E2 1267.982} C_VEL
LIN {X 0,Y 246.52,Z 707.548,A -85,B 0,C 180,E1 1266.421,E2 1266.421} C_VEL
LIN {X 0,Y 233.711,Z 723.066,A -85,B 0,C 180,E1 1264.55,E2 1264.55} C_VEL
LIN {X 0,Y 219.583,Z 738.108,A -85,B 0,C 180,E1 1262.158,E2 1262.158} C_VEL
LIN {X 0,Y 204.997,Z 751.737,A -85,B 0,C 180,E1 1259.249,E2 1259.249} C_VEL
LIN {X 0,Y 190.502,Z 763.778,A -85,B 0,C 180,E1 1255.762,E2 1255.762} C_VEL
LIN {X 0,Y 175.054,Z 775.053,A -85,B 0,C 180,E1 1251.132,E2 1251.132} C_VEL
LIN {X 0,Y 160.979,Z 784.15,A -85,B 0,C 180,E1 1245.693,E2 1245.693} C_VEL
LIN {X 0,Y 148.57,Z 791.382,A -85,B 0,C 180,E1 1239.311,E2 1239.311} C_VEL
LIN {X 0,Y 137.478,Z 797.237,A -85,B 0,C 180,E1 1231.318,E2 1231.318} C_VEL
LIN {X 0,Y 129.517,Z 801.086,A -85,B 0,C 180,E1 1222.676,E2 1222.676} C_VEL
LIN {X 0,Y 124.189,Z 803.354,A -85,B 0,C 180,E1 1212.898,E2 1212.898} C_VEL
LIN {X 0,Y 121.807,Z 803.88,A -85,B 0,C 180,E1 1203.371,E2 1203.371} C_VEL
LIN {X 0,Y 121.276,Z 803.25,A -85,B 0,C 180,E1 1194.869,E2 1194.869} C_VEL
LIN {X 0,Y 121.855,Z 801.535,A -85,B 0,C 180,E1 1186.694,E2 1186.694} C_VEL
LIN {X 0,Y 124.267,Z 798.248,A -85,B 0,C 180,E1 1177.401,E2 1177.401} C_VEL
LIN {X 0,Y 129.017,Z 793.391,A -85,B 0,C 180,E1 1168.476,E2 1168.476} C_VEL
LIN {X 0,Y 136.52,Z 786.399,A -85,B 0,C 180,E1 1159.881,E2 1159.881} C_VEL
LIN {X 0,Y 145.501,Z 778.162,A -85,B 0,C 180,E1 1152.818,E2 1152.818} C_VEL
LIN {X 0,Y 156.167,Z 768.086,A -85,B 0,C 180,E1 1146.617,E2 1146.617} C_VEL
LIN {X 0,Y 167.553,Z 756.624,A -85,B 0,C 180,E1 1141.489,E2 1141.489} C_VEL
LIN {X 0,Y 179.258,Z 743.815,A -85,B 0,C 180,E1 1137.25,E2 1137.25} C_VEL
LIN {X 0,Y 191.704,Z 728.61,A -85,B 0,C 180,E1 1133.522,E2 1133.522} C_VEL
LIN {X 0,Y 203.2,Z 712.751,A -85,B 0,C 180,E1 1130.603,E2 1130.603} C_VEL
LIN {X 0,Y 213.885,Z 696.013,A -85,B 0,C 180,E1 1128.234,E2 1128.234} C_VEL
LIN {X 0,Y 224.484,Z 676.849,A -85,B 0,C 180,E1 1126.15,E2 1126.15} C_VEL
LIN {X 0,Y 233.535,Z 657.557,A -85,B 0,C 180,E1 1124.537,E2 1124.537} C_VEL
LIN {X 0,Y 241.056,Z 638.421,A -85,B 0,C 180,E1 1123.29,E2 1123.29} C_VEL
LIN {X 0,Y 248.001,Z 616.279,A -85,B 0,C 180,E1 1122.203,E2 1122.203} C_VEL
LIN {X 0,Y 253.215,Z 594.109,A -85,B 0,C 180,E1 1121.417,E2 1121.417} C_VEL
LIN {X 0,Y 256.707,Z 572.414,A -85,B 0,C 180,E1 1120.882,E2 1120.882} C_VEL
LIN {X 0,Y 269.002,Z 464.156,A -85,B 0,C 180,E1 1118.787,E2 1118.787} C_VEL
LIN {X 0,Y 265.552,Z 456.79,A -85,B 0,C 180,E1 1115.503,E2 1115.503} C_VEL
LIN {X 0,Y 262.304,Z 450.26,A -85,B 0,C 180,E1 1111.735,E2 1111.735} C_VEL
LIN {X 0,Y 260.137,Z 446.136,A -85,B 0,C 180,E1 1108.587,E2 1108.587} C_VEL
LIN {X 0,Y 258.394,Z 442.717,A -85,B 0,C 180,E1 1105.189,E2 1105.189} C_VEL
LIN {X 0,Y 256.763,Z 439.216,A -85,B 0,C 180,E1 1099.327,E2 1099.327} C_VEL
LIN {X 0,Y 256.789,Z 439.202,A -85,B 0,C 180,E1 1093.508,E2 1093.508} C_VEL
LIN {X 0,Y 257.385,Z 440.758,A -85,B 0,C 180,E1 1090.518,E2 1090.518} C_VEL
LIN {X 0,Y 259.175,Z 443.832,A -85,B 0,C 180,E1 1086.088,E2 1086.088} C_VEL
LIN {X 0,Y 261.471,Z 448.137,A -85,B 0,C 180,E1 1082.299,E2 1082.299} C_VEL
LIN {X 0,Y 264.162,Z 453.259,A -85,B 0,C 180,E1 1078.914,E2 1078.914} C_VEL
LIN {X 0,Y 267.574,Z 459.782,A -85,B 0,C 180,E1 1075.444,E2 1075.444} C_VEL
LIN {X 0,Y 271.892,Z 468.696,A -85,B 0,C 180,E1 1071.763,E2 1071.763} C_VEL
LIN {X 0,Y 258.491,Z 591.372,A -85,B 0,C 180,E1 1069.394,E2 1069.394} C_VEL
LIN {X 0,Y 256.205,Z 604.606,A -85,B 0,C 180,E1 1069.064,E2 1069.064} C_VEL
LIN {X 0,Y 254.193,Z 612.091,A -85,B 0,C 180,E1 1069.081,E2 1069.081} C_VEL
LIN {X 0,Y 247.068,Z 630.684,A -85,B 0,C 180,E1 1069.787,E2 1069.787} C_VEL
LIN {X 0,Y 244.473,Z 638.018,A -85,B 0,C 180,E1 1069.711,E2 1069.711} C_VEL
LIN {X 0,Y 237.033,Z 658.486,A -85,B 0,C 180,E1 1068.782,E2 1068.782} C_VEL
LIN {X 0,Y 228.304,Z 678.34,A -85,B 0,C 180,E1 1067.573,E2 1067.573} C_VEL
LIN {X 0,Y 218.398,Z 697.413,A -85,B 0,C 180,E1 1066.051,E2 1066.051} C_VEL
LIN {X 0,Y 207.364,Z 715.697,A -85,B 0,C 180,E1 1064.129,E2 1064.129} C_VEL
LIN {X 0,Y 195.368,Z 732.931,A -85,B 0,C 180,E1 1061.72,E2 1061.72} C_VEL
LIN {X 0,Y 182.887,Z 748.844,A -85,B 0,C 180,E1 1058.754,E2 1058.754} C_VEL
LIN {X 0,Y 169.855,Z 763.741,A -85,B 0,C 180,E1 1055.02,E2 1055.02} C_VEL
LIN {X 0,Y 157.29,Z 776.821,A -85,B 0,C 180,E1 1050.552,E2 1050.552} C_VEL
LIN {X 0,Y 144.552,Z 789.056,A -85,B 0,C 180,E1 1044.698,E2 1044.698} C_VEL
LIN {X 0,Y 133.514,Z 799.154,A -85,B 0,C 180,E1 1037.843,E2 1037.843} C_VEL
LIN {X 0,Y 124.153,Z 807.795,A -85,B 0,C 180,E1 1029.504,E2 1029.504} C_VEL
LIN {X 0,Y 117.507,Z 814.571,A -85,B 0,C 180,E1 1020.128,E2 1020.128} C_VEL
LIN {X 0,Y 113.782,Z 819.534,A -85,B 0,C 180,E1 1010.036,E2 1010.036} C_VEL
LIN {X 0,Y 112.785,Z 822.636,A -85,B 0,C 180,E1 1000.207,E2 1000.207} C_VEL
LIN {X 0,Y 113.086,Z 823.943,A -85,B 0,C 180,E1 993.036,E2 993.036} C_VEL
LIN {X 0,Y 113.107,Z 824.32,A -85,B 0,C 180,E1 987.968,E2 987.968} C_VEL
LIN {X 0,Y 112.71,Z 824.05,A -85,B 0,C 180,E1 980.806,E2 980.806} C_VEL
LIN {X 0,Y 113.457,Z 822.509,A -85,B 0,C 180,E1 970.964,E2 970.964} C_VEL
LIN {X 0,Y 117.196,Z 819.185,A -85,B 0,C 180,E1 960.336,E2 960.336} C_VEL
LIN {X 0,Y 125.072,Z 813.803,A -85,B 0,C 180,E1 949.638,E2 949.638} C_VEL
LIN {X 0,Y 135.975,Z 806.874,A -85,B 0,C 180,E1 940.76,E2 940.76} C_VEL
LIN {X 0,Y 149.973,Z 797.756,A -85,B 0,C 180,E1 933.143,E2 933.143} C_VEL
LIN {X 0,Y 164.532,Z 787.639,A -85,B 0,C 180,E1 927.465,E2 927.465} C_VEL
LIN {X 0,Y 180.236,Z 775.848,A -85,B 0,C 180,E1 922.853,E2 922.853} C_VEL
LIN {X 0,Y 195.944,Z 762.847,A -85,B 0,C 180,E1 919.256,E2 919.256} C_VEL
LIN {X 0,Y 211.562,Z 748.354,A -85,B 0,C 180,E1 916.376,E2 916.376} C_VEL
LIN {X 0,Y 226.337,Z 732.918,A -85,B 0,C 180,E1 914.143,E2 914.143} C_VEL
LIN {X 0,Y 240.993,Z 715.524,A -85,B 0,C 180,E1 912.286,E2 912.286} C_VEL
LIN {X 0,Y 253.969,Z 697.902,A -85,B 0,C 180,E1 910.895,E2 910.895} C_VEL
LIN {X 0,Y 261.551,Z 686.214,A -85,B 0,C 180,E1 910.163,E2 910.163} C_VEL
LIN {X 0,Y 249.459,Z 703.534,A -85,B 0,C 180,E1 908.762,E2 908.762} C_VEL
LIN {X 0,Y 236.273,Z 719.807,A -85,B 0,C 180,E1 907.051,E2 907.051} C_VEL
LIN {X 0,Y 222.01,Z 735.169,A -85,B 0,C 180,E1 904.911,E2 904.911} C_VEL
LIN {X 0,Y 206.693,Z 749.423,A -85,B 0,C 180,E1 902.22,E2 902.22} C_VEL
LIN {X 0,Y 191.943,Z 761.485,A -85,B 0,C 180,E1 899.107,E2 899.107} C_VEL
LIN {X 0,Y 175.691,Z 773.206,A -85,B 0,C 180,E1 894.857,E2 894.857} C_VEL
LIN {X 0,Y 160.544,Z 782.809,A -85,B 0,C 180,E1 889.76,E2 889.76} C_VEL
LIN {X 0,Y 146.9,Z 790.525,A -85,B 0,C 180,E1 883.691,E2 883.691} C_VEL
LIN {X 0,Y 134.143,Z 796.915,A -85,B 0,C 180,E1 875.802,E2 875.802} C_VEL
LIN {X 0,Y 124.338,Z 801.221,A -85,B 0,C 180,E1 866.76,E2 866.76} C_VEL
LIN {X 0,Y 117.795,Z 803.719,A -85,B 0,C 180,E1 856.891,E2 856.891} C_VEL
LIN {X 0,Y 114.323,Z 804.632,A -85,B 0,C 180,E1 846.434,E2 846.434} C_VEL
LIN {X 0,Y 113.354,Z 804.257,A -85,B 0,C 180,E1 837.878,E2 837.878} C_VEL
LIN {X 0,Y 113.59,Z 802.876,A -85,B 0,C 180,E1 829.013,E2 829.013} C_VEL
LIN {X 0,Y 115.314,Z 800.276,A -85,B 0,C 180,E1 819.992,E2 819.992} C_VEL
LIN {X 0,Y 119.726,Z 795.747,A -85,B 0,C 180,E1 810.005,E2 810.005} C_VEL
LIN {X 0,Y 126.753,Z 789.545,A -85,B 0,C 180,E1 800.928,E2 800.928} C_VEL
LIN {X 0,Y 135.771,Z 781.875,A -85,B 0,C 180,E1 793.193,E2 793.193} C_VEL
LIN {X 0,Y 146.908,Z 772.04,A -85,B 0,C 180,E1 786.329,E2 786.329} C_VEL
LIN {X 0,Y 158.457,Z 761.146,A -85,B 0,C 180,E1 780.935,E2 780.935} C_VEL
LIN {X 0,Y 171.063,Z 748.194,A -85,B 0,C 180,E1 776.275,E2 776.275} C_VEL
LIN {X 0,Y 183.762,Z 733.693,A -85,B 0,C 180,E1 772.459,E2 772.459} C_VEL
LIN {X 0,Y 195.476,Z 718.698,A -85,B 0,C 180,E1 769.493,E2 769.493} C_VEL
LIN {X 0,Y 207.227,Z 701.585,A -85,B 0,C 180,E1 766.922,E2 766.922} C_VEL
LIN {X 0,Y 217.927,Z 683.501,A -85,B 0,C 180,E1 764.863,E2 764.863} C_VEL
LIN {X 0,Y 227.178,Z 665.218,A -85,B 0,C 180,E1 763.252,E2 763.252} C_VEL
LIN {X 0,Y 235.57,Z 645.54,A -85,B 0,C 180,E1 761.904,E2 761.904} C_VEL
LIN {X 0,Y 242.547,Z 625.579,A -85,B 0,C 180,E1 760.853,E2 760.853} C_VEL
LIN {X 0,Y 248.389,Z 604.294,A -85,B 0,C 180,E1 760.013,E2 760.013} C_VEL
LIN {X 0,Y 252.802,Z 581.902,A -85,B 0,C 180,E1 759.383,E2 759.383} C_VEL
LIN {X 0,Y 260.597,Z 516.817,A -85,B 0,C 180,E1 758.141,E2 758.141} C_VEL
LIN {X 0,Y 266.056,Z 469.116,A -85,B 0,C 180,E1 757.23,E2 757.23} C_VEL
LIN {X 0,Y 262.767,Z 461.845,A -85,B 0,C 180,E1 753.746,E2 753.746} C_VEL
LIN {X 0,Y 260.055,Z 456.439,A -85,B 0,C 180,E1 750.24,E2 750.24} C_VEL
LIN {X 0,Y 258.687,Z 453.637,A -85,B 0,C 180,E1 748.007,E2 748.007} C_VEL
LIN {X 0,Y 257.255,Z 450.626,A -85,B 0,C 180,E1 745.062,E2 745.062} C_VEL
LIN {X 0,Y 255.672,Z 447.123,A -85,B 0,C 180,E1 739.175,E2 739.175} C_VEL
LIN {X 0,Y 255.759,Z 447.192,A -85,B 0,C 180,E1 733.249,E2 733.249} C_VEL
LIN {X 0,Y 257.911,Z 451.56,A -85,B 0,C 180,E1 726.453,E2 726.453} C_VEL
LIN {X 0,Y 260.126,Z 455.898,A -85,B 0,C 180,E1 722.642,E2 722.642} C_VEL
LIN {X 0,Y 262.657,Z 460.876,A -85,B 0,C 180,E1 719.344,E2 719.344} C_VEL
LIN {X 0,Y 266.196,Z 467.911,A -85,B 0,C 180,E1 715.636,E2 715.636} C_VEL
LIN {X 0,Y 268.777,Z 473.749,A -85,B 0,C 180,E1 713.277,E2 713.277} C_VEL
LIN {X 0,Y 255.707,Z 590.858,A -85,B 0,C 180,E1 711.073,E2 711.073} C_VEL
LIN {X 0,Y 251.435,Z 613.007,A -85,B 0,C 180,E1 710.513,E2 710.513} C_VEL
LIN {X 0,Y 245.556,Z 634.508,A -85,B 0,C 180,E1 709.836,E2 709.836} C_VEL
LIN {X 0,Y 244.473,Z 638.018,A -85,B 0,C 180,E1 709.711,E2 709.711} C_VEL
LIN {X 0,Y 241.696,Z 645.269,A -85,B 0,C 180,E1 709.644,E2 709.644} C_VEL
LIN {X 0,Y 232.403,Z 663.157,A -85,B 0,C 180,E1 710.117,E2 710.117} C_VEL
LIN {X 0,Y 228.985,Z 669.947,A -85,B 0,C 180,E1 709.949,E2 709.949} C_VEL
LIN {X 0,Y 219.277,Z 689.488,A -85,B 0,C 180,E1 708.607,E2 708.607} C_VEL
LIN {X 0,Y 208.37,Z 708.224,A -85,B 0,C 180,E1 706.913,E2 706.913} C_VEL
LIN {X 0,Y 196.801,Z 725.485,A -85,B 0,C 180,E1 704.85,E2 704.85} C_VEL
LIN {X 0,Y 184.033,Z 742.053,A -85,B 0,C 180,E1 702.195,E2 702.195} C_VEL
LIN {X 0,Y 171.314,Z 756.744,A -85,B 0,C 180,E1 699.027,E2 699.027} C_VEL
LIN {X 0,Y 157.715,Z 770.91,A -85,B 0,C 180,E1 694.862,E2 694.862} C_VEL
LIN {X 0,Y 145.354,Z 782.727,A -85,B 0,C 180,E1 690.071,E2 690.071} C_VEL
LIN {X 0,Y 132.789,Z 793.832,A -85,B 0,C 180,E1 683.667,E2 683.667} C_VEL
LIN {X 0,Y 122.105,Z 802.951,A -85,B 0,C 180,E1 676.095,E2 676.095} C_VEL
LIN {X 0,Y 113.049,Z 810.951,A -85,B 0,C 180,E1 666.399,E2 666.399} C_VEL
LIN {X 0,Y 107.436,Z 816.801,A -85,B 0,C 180,E1 655.932,E2 655.932} C_VEL
LIN {X 0,Y 105.049,Z 820.628,A -85,B 0,C 180,E1 645.45,E2 645.45} C_VEL
LIN {X 0,Y 104.986,Z 822.894,A -85,B 0,C 180,E1 635.459,E2 635.459} C_VEL
LIN {X 0,Y 105.194,Z 823.556,A -85,B 0,C 180,E1 629.45,E2 629.45} C_VEL
LIN {X 0,Y 104.785,Z 823.54,A -85,B 0,C 180,E1 622.317,E2 622.317} C_VEL
LIN {X 0,Y 105.301,Z 822.232,A -85,B 0,C 180,E1 611.73,E2 611.73} C_VEL
LIN {X 0,Y 109.223,Z 819.176,A -85,B 0,C 180,E1 599.763,E2 599.763} C_VEL
LIN {X 0,Y 117.475,Z 814.158,A -85,B 0,C 180,E1 588.398,E2 588.398} C_VEL
LIN {X 0,Y 128.895,Z 807.484,A -85,B 0,C 180,E1 579.124,E2 579.124} C_VEL
LIN {X 0,Y 143.069,Z 799.018,A -85,B 0,C 180,E1 571.496,E2 571.496} C_VEL
LIN {X 0,Y 159.321,Z 788.599,A -85,B 0,C 180,E1 565.343,E2 565.343} C_VEL
LIN {X 0,Y 175.45,Z 777.273,A -85,B 0,C 180,E1 560.828,E2 560.828} C_VEL
LIN {X 0,Y 191.697,Z 764.51,A -85,B 0,C 180,E1 557.298,E2 557.298} C_VEL
LIN {X 0,Y 207.913,Z 750.228,A -85,B 0,C 180,E1 554.484,E2 554.484} C_VEL
LIN {X 0,Y 224.512,Z 733.653,A -85,B 0,C 180,E1 552.157,E2 552.157} C_VEL
LIN {X 0,Y 238.961,Z 717.197,A -85,B 0,C 180,E1 550.48,E2 550.48} C_VEL
LIN {X 0,Y 243.588,Z 711.393,A -85,B 0,C 180,E1 549.989,E2 549.989} C_VEL
LIN {X 0,Y 229.81,Z 727.085,A -85,B 0,C 180,E1 548.257,E2 548.257} C_VEL
LIN {X 0,Y 214.729,Z 741.858,A -85,B 0,C 180,E1 546.063,E2 546.063} C_VEL
LIN {X 0,Y 199.331,Z 755.063,A -85,B 0,C 180,E1 543.403,E2 543.403} C_VEL
LIN {X 0,Y 182.483,Z 767.677,A -85,B 0,C 180,E1 539.846,E2 539.846} C_VEL
LIN {X 0,Y 167.423,Z 777.567,A -85,B 0,C 180,E1 535.852,E2 535.852} C_VEL
LIN {X 0,Y 151.817,Z 786.567,A -85,B 0,C 180,E1 530.526,E2 530.526} C_VEL
LIN {X 0,Y 137.393,Z 793.798,A -85,B 0,C 180,E1 523.878,E2 523.878} C_VEL
LIN {X 0,Y 125.267,Z 799.13,A -85,B 0,C 180,E1 515.984,E2 515.984} C_VEL
LIN {X 0,Y 115.421,Z 802.928,A -85,B 0,C 180,E1 506.274,E2 506.274} C_VEL
LIN {X 0,Y 109.082,Z 804.963,A -85,B 0,C 180,E1 495.647,E2 495.647} C_VEL
LIN {X 0,Y 106.048,Z 805.371,A -85,B 0,C 180,E1 484.897,E2 484.897} C_VEL
LIN {X 0,Y 105.329,Z 804.64,A -85,B 0,C 180,E1 475.294,E2 475.294} C_VEL
LIN {X 0,Y 105.908,Z 803.007,A -85,B 0,C 180,E1 466.458,E2 466.458} C_VEL
LIN {X 0,Y 108.665,Z 799.735,A -85,B 0,C 180,E1 455.815,E2 455.815} C_VEL
LIN {X 0,Y 114.351,Z 794.727,A -85,B 0,C 180,E1 445.492,E2 445.492} C_VEL
LIN {X 0,Y 122.735,Z 787.913,A -85,B 0,C 180,E1 436.34,E2 436.34} C_VEL
LIN {X 0,Y 133.083,Z 779.509,A -85,B 0,C 180,E1 428.677,E2 428.677} C_VEL
LIN {X 0,Y 144.653,Z 769.662,A -85,B 0,C 180,E1 422.417,E2 422.417} C_VEL
LIN {X 0,Y 157.081,Z 758.242,A -85,B 0,C 180,E1 417.25,E2 417.25} C_VEL
LIN {X 0,Y 169.702,Z 745.465,A -85,B 0,C 180,E1 413.066,E2 413.066} C_VEL
LIN {X 0,Y 182.717,Z 730.615,A -85,B 0,C 180,E1 409.515,E2 409.515} C_VEL
LIN {X 0,Y 194.758,Z 715.067,A -85,B 0,C 180,E1 406.74,E2 406.74} C_VEL
LIN {X 0,Y 206.423,Z 697.865,A -85,B 0,C 180,E1 404.407,E2 404.407} C_VEL
LIN {X 0,Y 217.06,Z 679.719,A -85,B 0,C 180,E1 402.527,E2 402.527} C_VEL
LIN {X 0,Y 226.55,Z 660.717,A -85,B 0,C 180,E1 401.006,E2 401.006} C_VEL
LIN {X 0,Y 234.81,Z 640.753,A -85,B 0,C 180,E1 399.777,E2 399.777} C_VEL
LIN {X 0,Y 241.584,Z 620.38,A -85,B 0,C 180,E1 398.824,E2 398.824} C_VEL
LIN {X 0,Y 247.112,Z 598.859,A -85,B 0,C 180,E1 398.077,E2 398.077} C_VEL
LIN {X 0,Y 251.241,Z 575.887,A -85,B 0,C 180,E1 397.519,E2 397.519} C_VEL
LIN {X 0,Y 263.32,Z 474.139,A -85,B 0,C 180,E1 395.656,E2 395.656} C_VEL
LIN {X 0,Y 260.302,Z 467.579,A -85,B 0,C 180,E1 392.138,E2 392.138} C_VEL
LIN {X 0,Y 257.762,Z 462.002,A -85,B 0,C 180,E1 388.299,E2 388.299} C_VEL
LIN {X 0,Y 256.022,Z 458.387,A -85,B 0,C 180,E1 384.698,E2 384.698} C_VEL
LIN {X 0,Y 254.582,Z 455.031,A -85,B 0,C 180,E1 379.023,E2 379.023} C_VEL
LIN {X 0,Y 254.696,Z 455.137,A -85,B 0,C 180,E1 373.215,E2 373.215} C_VEL
LIN {X 0,Y 256.644,Z 459.286,A -85,B 0,C 180,E1 366.822,E2 366.822} C_VEL
LIN {X 0,Y 258.788,Z 463.657,A -85,B 0,C 180,E1 362.988,E2 362.988} C_VEL
LIN {X 0,Y 261.338,Z 468.845,A -85,B 0,C 180,E1 359.56,E2 359.56} C_VEL
LIN {X 0,Y 264.575,Z 475.643,A -85,B 0,C 180,E1 356.056,E2 356.056} C_VEL
LIN {X 0,Y 265.817,Z 478.678,A -85,B 0,C 180,E1 354.826,E2 354.826} C_VEL
LIN {X 0,Y 252.994,Z 590.767,A -85,B 0,C 180,E1 352.771,E2 352.771} C_VEL
LIN {X 0,Y 248.61,Z 613.037,A -85,B 0,C 180,E1 352.229,E2 352.229} C_VEL
LIN {X 0,Y 242.806,Z 633.911,A -85,B 0,C 180,E1 351.603,E2 351.603} C_VEL
LIN {X 0,Y 235.037,Z 655.723,A -85,B 0,C 180,E1 350.709,E2 350.709} C_VEL
LIN {X 0,Y 228.985,Z 669.947,A -85,B 0,C 180,E1 349.949,E2 349.949} C_VEL
LIN {X 0,Y 225.414,Z 676.813,A -85,B 0,C 180,E1 349.754,E2 349.754} C_VEL
LIN {X 0,Y 213.598,Z 694.453,A -85,B 0,C 180,E1 349.972,E2 349.972} C_VEL
LIN {X 0,Y 209.997,Z 699.939,A -85,B 0,C 180,E1 349.688,E2 349.688} C_VEL
LIN {X 0,Y 197.937,Z 718.514,A -85,B 0,C 180,E1 347.79,E2 347.79} C_VEL
LIN {X 0,Y 185.819,Z 734.814,A -85,B 0,C 180,E1 345.576,E2 345.576} C_VEL
LIN {X 0,Y 172.315,Z 750.741,A -85,B 0,C 180,E1 342.638,E2 342.638} C_VEL
LIN {X 0,Y 159.335,Z 764.331,A -85,B 0,C 180,E1 339.217,E2 339.217} C_VEL
LIN {X 0,Y 145.101,Z 777.791,A -85,B 0,C 180,E1 334.503,E2 334.503} C_VEL
LIN {X 0,Y 132.032,Z 789.135,A -85,B 0,C 180,E1 328.83,E2 328.83} C_VEL
LIN {X 0,Y 119.869,Z 799.038,A -85,B 0,C 180,E1 321.627,E2 321.627} C_VEL
LIN {X 0,Y 109.861,Z 807.029,A -85,B 0,C 180,E1 313.038,E2 313.038} C_VEL
LIN {X 0,Y 101.909,Z 813.915,A -85,B 0,C 180,E1 301.985,E2 301.985} C_VEL
LIN {X 0,Y 97.778,Z 818.693,A -85,B 0,C 180,E1 290.339,E2 290.339} C_VEL
LIN {X 0,Y 96.846,Z 821.428,A -85,B 0,C 180,E1 279.502,E2 279.502} C_VEL
LIN {X 0,Y 97.205,Z 822.554,A -85,B 0,C 180,E1 271.762,E2 271.762} C_VEL
LIN {X 0,Y 97.044,Z 822.835,A -85,B 0,C 180,E1 265.858,E2 265.858} C_VEL
LIN {X 0,Y 96.793,Z 822.412,A -85,B 0,C 180,E1 256.858,E2 256.858} C_VEL
LIN {X 0,Y 99.11,Z 820.431,A -85,B 0,C 180,E1 244.285,E2 244.285} C_VEL
LIN {X 0,Y 106.032,Z 816.472,A -85,B 0,C 180,E1 231.504,E2 231.504} C_VEL
LIN {X 0,Y 117.206,Z 810.579,A -85,B 0,C 180,E1 220.596,E2 220.596} C_VEL
LIN {X 0,Y 131.066,Z 803.156,A -85,B 0,C 180,E1 212.129,E2 212.129} C_VEL
LIN {X 0,Y 147.225,Z 793.9,A -85,B 0,C 180,E1 205.403,E2 205.403} C_VEL
LIN {X 0,Y 164.246,Z 783.165,A -85,B 0,C 180,E1 200.306,E2 200.306} C_VEL
LIN {X 0,Y 181.399,Z 771.001,A -85,B 0,C 180,E1 196.439,E2 196.439} C_VEL
LIN {X 0,Y 197.508,Z 758.154,A -85,B 0,C 180,E1 193.586,E2 193.586} C_VEL
LIN {X 0,Y 214.076,Z 743.307,A -85,B 0,C 180,E1 191.229,E2 191.229} C_VEL
LIN {X 0,Y 225.538,Z 731.746,A -85,B 0,C 180,E1 189.82,E2 189.82} C_VEL
LIN {X 0,Y 210.936,Z 745.382,A -85,B 0,C 180,E1 187.811,E2 187.811} C_VEL
LIN {X 0,Y 194.776,Z 758.466,A -85,B 0,C 180,E1 185.178,E2 185.178} C_VEL
LIN {X 0,Y 178.46,Z 769.935,A -85,B 0,C 180,E1 181.929,E2 181.929} C_VEL
LIN {X 0,Y 162.103,Z 779.984,A -85,B 0,C 180,E1 177.815,E2 177.815} C_VEL
LIN {X 0,Y 145.976,Z 788.602,A -85,B 0,C 180,E1 172.526,E2 172.526} C_VEL
LIN {X 0,Y 130.984,Z 795.568,A -85,B 0,C 180,E1 165.817,E2 165.817} C_VEL
LIN {X 0,Y 117.261,Z 800.99,A -85,B 0,C 180,E1 156.911,E2 156.911} C_VEL
LIN {X 0,Y 107.136,Z 804.308,A -85,B 0,C 180,E1 146.596,E2 146.596} C_VEL
LIN {X 0,Y 100.627,Z 805.93,A -85,B 0,C 180,E1 134.876,E2 134.876} C_VEL
LIN {X 0,Y 97.784,Z 805.988,A -85,B 0,C 180,E1 122.822,E2 122.822} C_VEL
LIN {X 0,Y 97.389,Z 804.957,A -85,B 0,C 180,E1 112.969,E2 112.969} C_VEL
LIN {X 0,Y 98.64,Z 802.805,A -85,B 0,C 180,E1 102.296,E2 102.296} C_VEL
LIN {X 0,Y 102.559,Z 799.008,A -85,B 0,C 180,E1 91.123,E2 91.123} C_VEL
LIN {X 0,Y 109.334,Z 793.638,A -85,B 0,C 180,E1 80.955,E2 80.955} C_VEL
LIN {X 0,Y 119.501,Z 786.013,A -85,B 0,C 180,E1 71.467,E2 71.467} C_VEL
LIN {X 0,Y 130.871,Z 777.251,A -85,B 0,C 180,E1 64.189,E2 64.189} C_VEL
LIN {X 0,Y 143.79,Z 766.57,A -85,B 0,C 180,E1 58.103,E2 58.103} C_VEL
LIN {X 0,Y 157.328,Z 754.158,A -85,B 0,C 180,E1 53.197,E2 53.197} C_VEL
LIN {X 0,Y 170.458,Z 740.688,A -85,B 0,C 180,E1 49.381,E2 49.381} C_VEL
LIN {X 0,Y 183.551,Z 725.56,A -85,B 0,C 180,E1 46.232,E2 46.232} C_VEL
LIN {X 0,Y 196.187,Z 708.887,A -85,B 0,C 180,E1 43.645,E2 43.645} C_VEL
LIN {X 0,Y 207.383,Z 691.913,A -85,B 0,C 180,E1 41.648,E2 41.648} C_VEL
LIN {X 0,Y 217.874,Z 673.343,A -85,B 0,C 180,E1 39.974,E2 39.974} C_VEL
LIN {X 0,Y 227.144,Z 653.747,A -85,B 0,C 180,E1 38.622,E2 38.622} C_VEL
LIN {X 0,Y 234.689,Z 634.431,A -85,B 0,C 180,E1 37.592,E2 37.592} C_VEL
LIN {X 0,Y 241.497,Z 612.565,A -85,B 0,C 180,E1 36.713,E2 36.713} C_VEL
LIN {X 0,Y 246.504,Z 591.06,A -85,B 0,C 180,E1 36.086,E2 36.086} C_VEL
LIN {X 0,Y 250.012,Z 568.675,A -85,B 0,C 180,E1 35.624,E2 35.624} C_VEL
LIN {X 0,Y 260.676,Z 479.368,A -85,B 0,C 180,E1 34.053,E2 34.053} C_VEL
LIN {X 0,Y 257.74,Z 472.743,A -85,B 0,C 180,E1 30.154,E2 30.154} C_VEL
LIN {X 0,Y 256.009,Z 468.988,A -85,B 0,C 180,E1 27.188,E2 27.188} C_VEL
LIN {X 0,Y 254.779,Z 466.146,A -85,B 0,C 180,E1 24.332,E2 24.332} C_VEL
LIN {X 0,Y 253.486,Z 462.93,A -85,B 0,C 180,E1 18.807,E2 18.807} C_VEL
LIN {X 0,Y 253.631,Z 463.092,A -85,B 0,C 180,E1 13.179,E2 13.179} C_VEL
LIN {X 0,Y 255.428,Z 467.141,A -85,B 0,C 180,E1 7.081,E2 7.081} C_VEL
LIN {X 0,Y 257.402,Z 471.327,A -85,B 0,C 180,E1 3.397,E2 3.397} C_VEL
LIN {X 0,Y 260.015,Z 476.804,A -85,B 0,C 180,E1 -0.222,E2 -0.222} C_VEL
LIN {X 0,Y 263.019,Z 483.519,A -85,B 0,C 180,E1 -3.586,E2 -3.586} C_VEL
LIN {X 0,Y 250.57,Z 590.218,A -85,B 0,C 180,E1 -5.488,E2 -5.488} C_VEL
LIN {X 0,Y 246.13,Z 612.452,A -85,B 0,C 180,E1 -6.004,E2 -6.004} C_VEL
LIN {X 0,Y 240.291,Z 633.22,A -85,B 0,C 180,E1 -6.591,E2 -6.591} C_VEL
LIN {X 0,Y 232.585,Z 654.638,A -85,B 0,C 180,E1 -7.412,E2 -7.412} C_VEL
LIN {X 0,Y 223.835,Z 674.491,A -85,B 0,C 180,E1 -8.449,E2 -8.449} C_VEL
LIN {X 0,Y 213.578,Z 693.956,A -85,B 0,C 180,E1 -9.806,E2 -9.806} C_VEL
LIN {X 0,Y 209.997,Z 699.939,A -85,B 0,C 180,E1 -10.312,E2 -10.312} C_VEL
LIN {X 0,Y 205.673,Z 706.328,A -85,B 0,C 180,E1 -10.645,E2 -10.645} C_VEL
LIN {X 0,Y 192.687,Z 721.676,A -85,B 0,C 180,E1 -10.734,E2 -10.734} C_VEL
LIN {X 0,Y 187.821,Z 727.496,A -85,B 0,C 180,E1 -11.201,E2 -11.201} C_VEL
LIN {X 0,Y 174.62,Z 743.551,A -85,B 0,C 180,E1 -13.671,E2 -13.671} C_VEL
LIN {X 0,Y 160.822,Z 758.305,A -85,B 0,C 180,E1 -16.79,E2 -16.79} C_VEL
LIN {X 0,Y 146.709,Z 771.721,A -85,B 0,C 180,E1 -20.759,E2 -20.759} C_VEL
LIN {X 0,Y 132.272,Z 784.106,A -85,B 0,C 180,E1 -26.007,E2 -26.007} C_VEL
LIN {X 0,Y 119.018,Z 794.582,A -85,B 0,C 180,E1 -32.528,E2 -32.528} C_VEL
LIN {X 0,Y 107.105,Z 803.528,A -85,B 0,C 180,E1 -40.882,E2 -40.882} C_VEL
LIN {X 0,Y 97.536,Z 810.758,A -85,B 0,C 180,E1 -51.303,E2 -51.303} C_VEL
LIN {X 0,Y 91.391,Z 816.208,A -85,B 0,C 180,E1 -63.357,E2 -63.357} C_VEL
LIN {X 0,Y 88.982,Z 819.835,A -85,B 0,C 180,E1 -75.695,E2 -75.695} C_VEL
LIN {X 0,Y 89.135,Z 821.574,A -85,B 0,C 180,E1 -86.148,E2 -86.148} C_VEL
LIN {X 0,Y 89.202,Z 822.077,A -85,B 0,C 180,E1 -91.934,E2 -91.934} C_VEL
LIN {X 0,Y 88.773,Z 821.915,A -85,B 0,C 180,E1 -101.704,E2 -101.704} C_VEL
LIN {X 0,Y 90.492,Z 820.477,A -85,B 0,C 180,E1 -114.138,E2 -114.138} C_VEL
LIN {X 0,Y 97.127,Z 817.061,A -85,B 0,C 180,E1 -128.153,E2 -128.153} C_VEL
LIN {X 0,Y 107.82,Z 812.118,A -85,B 0,C 180,E1 -139.518,E2 -139.518} C_VEL
LIN {X 0,Y 122.932,Z 804.881,A -85,B 0,C 180,E1 -149.172,E2 -149.172} C_VEL
LIN {X 0,Y 139.836,Z 795.997,A -85,B 0,C 180,E1 -156.247,E2 -156.247} C_VEL
LIN {X 0,Y 157.219,Z 785.848,A -85,B 0,C 180,E1 -161.378,E2 -161.378} C_VEL
LIN {X 0,Y 175.651,Z 773.754,A -85,B 0,C 180,E1 -165.407,E2 -165.407} C_VEL
LIN {X 0,Y 193.907,Z 760.131,A -85,B 0,C 180,E1 -168.452,E2 -168.452} C_VEL
LIN {X 0,Y 207.573,Z 748.558,A -85,B 0,C 180,E1 -170.336,E2 -170.336} C_VEL
LIN {X 0,Y 191.386,Z 761.071,A -85,B 0,C 180,E1 -172.795,E2 -172.795} C_VEL
LIN {X 0,Y 174.002,Z 772.68,A -85,B 0,C 180,E1 -176.043,E2 -176.043} C_VEL
LIN {X 0,Y 156.987,Z 782.402,A -85,B 0,C 180,E1 -180.092,E2 -180.092} C_VEL
LIN {X 0,Y 140.327,Z 790.631,A -85,B 0,C 180,E1 -185.311,E2 -185.311} C_VEL
LIN {X 0,Y 123.911,Z 797.53,A -85,B 0,C 180,E1 -192.462,E2 -192.462} C_VEL
LIN {X 0,Y 110.401,Z 802.314,A -85,B 0,C 180,E1 -201.106,E2 -201.106} C_VEL
LIN {X 0,Y 99.376,Z 805.514,A -85,B 0,C 180,E1 -212.301,E2 -212.301} C_VEL
LIN {X 0,Y 92.677,Z 806.803,A -85,B 0,C 180,E1 -224.589,E2 -224.589} C_VEL
LIN {X 0,Y 89.821,Z 806.656,A -85,B 0,C 180,E1 -236.937,E2 -236.937} C_VEL
LIN {X 0,Y 89.411,Z 805.64,A -85,B 0,C 180,E1 -246.952,E2 -246.952} C_VEL
LIN {X 0,Y 90.786,Z 803.436,A -85,B 0,C 180,E1 -258.559,E2 -258.559} C_VEL
LIN {X 0,Y 95.129,Z 799.614,A -85,B 0,C 180,E1 -270.596,E2 -270.596} C_VEL
LIN {X 0,Y 102.454,Z 794.261,A -85,B 0,C 180,E1 -281.249,E2 -281.249} C_VEL
LIN {X 0,Y 112.925,Z 786.943,A -85,B 0,C 180,E1 -290.736,E2 -290.736} C_VEL
LIN {X 0,Y 124.928,Z 778.241,A -85,B 0,C 180,E1 -298.172,E2 -298.172} C_VEL
LIN {X 0,Y 138.445,Z 767.6,A -85,B 0,C 180,E1 -304.28,E2 -304.28} C_VEL
LIN {X 0,Y 152.286,Z 755.438,A -85,B 0,C 180,E1 -309.067,E2 -309.067} C_VEL
LIN {X 0,Y 166.066,Z 741.848,A -85,B 0,C 180,E1 -312.866,E2 -312.866} C_VEL
LIN {X 0,Y 179.898,Z 726.367,A -85,B 0,C 180,E1 -315.998,E2 -315.998} C_VEL
LIN {X 0,Y 192.475,Z 710.248,A -85,B 0,C 180,E1 -318.416,E2 -318.416} C_VEL
LIN {X 0,Y 203.916,Z 693.414,A -85,B 0,C 180,E1 -320.332,E2 -320.332} C_VEL
LIN {X 0,Y 215.061,Z 674.126,A -85,B 0,C 180,E1 -321.997,E2 -321.997} C_VEL
LIN {X 0,Y 224.505,Z 654.589,A -85,B 0,C 180,E1 -323.283,E2 -323.283} C_VEL
LIN {X 0,Y 232.183,Z 635.367,A -85,B 0,C 180,E1 -324.261,E2 -324.261} C_VEL
LIN {X 0,Y 238.985,Z 614.104,A -85,B 0,C 180,E1 -325.082,E2 -325.082} C_VEL
LIN {X 0,Y 244.141,Z 592.746,A -85,B 0,C 180,E1 -325.684,E2 -325.684} C_VEL
LIN {X 0,Y 247.814,Z 570.18,A -85,B 0,C 180,E1 -326.134,E2 -326.134} C_VEL
LIN {X 0,Y 258.204,Z 484.79,A -85,B 0,C 180,E1 -327.578,E2 -327.578} C_VEL
LIN {X 0,Y 255.814,Z 479.229,A -85,B 0,C 180,E1 -331.14,E2 -331.14} C_VEL
LIN {X 0,Y 254.437,Z 476.106,A -85,B 0,C 180,E1 -333.765,E2 -333.765} C_VEL
LIN {X 0,Y 253.477,Z 473.789,A -85,B 0,C 180,E1 -336.218,E2 -336.218} C_VEL
LIN {X 0,Y 252.407,Z 470.849,A -85,B 0,C 180,E1 -341.287,E2 -341.287} C_VEL
LIN {X 0,Y 252.548,Z 471.012,A -85,B 0,C 180,E1 -346.727,E2 -346.727} C_VEL
LIN {X 0,Y 254.217,Z 474.994,A -85,B 0,C 180,E1 -352.658,E2 -352.658} C_VEL
LIN {X 0,Y 256.032,Z 479.004,A -85,B 0,C 180,E1 -356.195,E2 -356.195} C_VEL
LIN {X 0,Y 258.649,Z 484.683,A -85,B 0,C 180,E1 -359.946,E2 -359.946} C_VEL
LIN {X 0,Y 260.32,Z 488.804,A -85,B 0,C 180,E1 -361.989,E2 -361.989} C_VEL
LIN {X 0,Y 248.257,Z 589.921,A -85,B 0,C 180,E1 -363.724,E2 -363.724} C_VEL
LIN {X 0,Y 243.737,Z 612.218,A -85,B 0,C 180,E1 -364.217,E2 -364.217} C_VEL
LIN {X 0,Y 237.776,Z 633.091,A -85,B 0,C 180,E1 -364.769,E2 -364.769} C_VEL
LIN {X 0,Y 230.025,Z 654.305,A -85,B 0,C 180,E1 -365.531,E2 -365.531} C_VEL
LIN {X 0,Y 221.276,Z 673.887,A -85,B 0,C 180,E1 -366.488,E2 -366.488} C_VEL
LIN {X 0,Y 210.888,Z 693.31,A -85,B 0,C 180,E1 -367.76,E2 -367.76} C_VEL
LIN {X 0,Y 199.595,Z 711.216,A -85,B 0,C 180,E1 -369.322,E2 -369.322} C_VEL
LIN {X 0,Y 187.821,Z 727.496,A -85,B 0,C 180,E1 -371.201,E2 -371.201} C_VEL
LIN {X 0,Y 182.83,Z 733.313,A -85,B 0,C 180,E1 -371.718,E2 -371.718} C_VEL
LIN {X 0,Y 168.228,Z 746.985,A -85,B 0,C 180,E1 -372.231,E2 -372.231} C_VEL
LIN {X 0,Y 162.806,Z 752.126,A -85,B 0,C 180,E1 -372.955,E2 -372.955} C_VEL
LIN {X 0,Y 148.042,Z 766.407,A -85,B 0,C 180,E1 -376.482,E2 -376.482} C_VEL
LIN {X 0,Y 133.725,Z 778.629,A -85,B 0,C 180,E1 -380.848,E2 -380.848} C_VEL
LIN {X 0,Y 119.588,Z 789.593,A -85,B 0,C 180,E1 -386.554,E2 -386.554} C_VEL
LIN {X 0,Y 106.226,Z 799.204,A -85,B 0,C 180,E1 -394.086,E2 -394.086} C_VEL
LIN {X 0,Y 94.543,Z 807.326,A -85,B 0,C 180,E1 -404.026,E2 -404.026} C_VEL
LIN {X 0,Y 86.126,Z 813.477,A -85,B 0,C 180,E1 -416.143,E2 -416.143} C_VEL
LIN {X 0,Y 81.654,Z 817.894,A -85,B 0,C 180,E1 -429.957,E2 -429.957} C_VEL
LIN {X 0,Y 80.945,Z 820.309,A -85,B 0,C 180,E1 -442.198,E2 -442.198} C_VEL
LIN {X 0,Y 81.325,Z 821.14,A -85,B 0,C 180,E1 -450.007,E2 -450.007} C_VEL
LIN {X 0,Y 80.871,Z 821.309,A -85,B 0,C 180,E1 -457.824,E2 -457.824} C_VEL
LIN {X 0,Y 81.842,Z 820.487,A -85,B 0,C 180,E1 -471.786,E2 -471.786} C_VEL
LIN {X 0,Y 87.458,Z 817.859,A -85,B 0,C 180,E1 -486.484,E2 -486.484} C_VEL
LIN {X 0,Y 98.411,Z 813.345,A -85,B 0,C 180,E1 -499.65,E2 -499.65} C_VEL
LIN {X 0,Y 113.32,Z 807.026,A -85,B 0,C 180,E1 -509.856,E2 -509.856} C_VEL
LIN {X 0,Y 130.14,Z 799.205,A -85,B 0,C 180,E1 -517.224,E2 -517.224} C_VEL
LIN {X 0,Y 148.639,Z 789.414,A -85,B 0,C 180,E1 -522.796,E2 -522.796} C_VEL
LIN {X 0,Y 166.448,Z 778.731,A -85,B 0,C 180,E1 -526.702,E2 -526.702} C_VEL
LIN {X 0,Y 184.919,Z 766.192,A -85,B 0,C 180,E1 -529.776,E2 -529.776} C_VEL
LIN {X 0,Y 189.588,Z 762.711,A -85,B 0,C 180,E1 -530.489,E2 -530.489} C_VEL
LIN {X 0,Y 172.107,Z 773.959,A -85,B 0,C 180,E1 -533.453,E2 -533.453} C_VEL
LIN {X 0,Y 153.121,Z 784.317,A -85,B 0,C 180,E1 -537.602,E2 -537.602} C_VEL
LIN {X 0,Y 136.124,Z 792.12,A -85,B 0,C 180,E1 -542.548,E2 -542.548} C_VEL
LIN {X 0,Y 119.545,Z 798.578,A -85,B 0,C 180,E1 -549.245,E2 -549.245} C_VEL
LIN {X 0,Y 104.231,Z 803.473,A -85,B 0,C 180,E1 -558.45,E2 -558.45} C_VEL
LIN {X 0,Y 92.573,Z 806.412,A -85,B 0,C 180,E1 -569.785,E2 -569.785} C_VEL
LIN {X 0,Y 85.022,Z 807.638,A -85,B 0,C 180,E1 -583.178,E2 -583.178} C_VEL
LIN {X 0,Y 81.858,Z 807.318,A -85,B 0,C 180,E1 -596.649,E2 -596.649} C_VEL
LIN {X 0,Y 81.493,Z 806.132,A -85,B 0,C 180,E1 -608.395,E2 -608.395} C_VEL
LIN {X 0,Y 83.303,Z 803.697,A -85,B 0,C 180,E1 -621.016,E2 -621.016} C_VEL
LIN {X 0,Y 88.504,Z 799.717,A -85,B 0,C 180,E1 -633.88,E2 -633.88} C_VEL
LIN {X 0,Y 97.633,Z 793.684,A -85,B 0,C 180,E1 -645.73,E2 -645.73} C_VEL
LIN {X 0,Y 109.059,Z 786.16,A -85,B 0,C 180,E1 -654.938,E2 -654.938} C_VEL
LIN {X 0,Y 122.081,Z 777.074,A -85,B 0,C 180,E1 -662.159,E2 -662.159} C_VEL
LIN {X 0,Y 135.687,Z 766.693,A -85,B 0,C 180,E1 -667.7,E2 -667.7} C_VEL
LIN {X 0,Y 150.194,Z 754.32,A -85,B 0,C 180,E1 -672.244,E2 -672.244} C_VEL
LIN {X 0,Y 164.508,Z 740.392,A -85,B 0,C 180,E1 -675.817,E2 -675.817} C_VEL
LIN {X 0,Y 177.959,Z 725.467,A -85,B 0,C 180,E1 -678.59,E2 -678.59} C_VEL
LIN {X 0,Y 191.247,Z 708.529,A -85,B 0,C 180,E1 -680.924,E2 -680.924} C_VEL
LIN {X 0,Y 203.406,Z 690.5,A -85,B 0,C 180,E1 -682.775,E2 -682.775} C_VEL
LIN {X 0,Y 213.876,Z 672.329,A -85,B 0,C 180,E1 -684.198,E2 -684.198} C_VEL
LIN {X 0,Y 223.739,Z 651.842,A -85,B 0,C 180,E1 -685.424,E2 -685.424} C_VEL
LIN {X 0,Y 231.776,Z 631.175,A -85,B 0,C 180,E1 -686.359,E2 -686.359} C_VEL
LIN {X 0,Y 238.138,Z 610.354,A -85,B 0,C 180,E1 -687.065,E2 -687.065} C_VEL
LIN {X 0,Y 243.094,Z 588.51,A -85,B 0,C 180,E1 -687.609,E2 -687.609} C_VEL
LIN {X 0,Y 247.116,Z 561.109,A -85,B 0,C 180,E1 -688.089,E2 -688.089} C_VEL
LIN {X 0,Y 255.865,Z 490.406,A -85,B 0,C 180,E1 -689.211,E2 -689.211} C_VEL
LIN {X 0,Y 253.735,Z 485.032,A -85,B 0,C 180,E1 -692.938,E2 -692.938} C_VEL
LIN {X 0,Y 252.322,Z 481.662,A -85,B 0,C 180,E1 -696.41,E2 -696.41} C_VEL
LIN {X 0,Y 251.322,Z 478.762,A -85,B 0,C 180,E1 -701.444,E2 -701.444} C_VEL
LIN {X 0,Y 251.47,Z 478.951,A -85,B 0,C 180,E1 -706.669,E2 -706.669} C_VEL
LIN {X 0,Y 252.967,Z 482.717,A -85,B 0,C 180,E1 -712.279,E2 -712.279} C_VEL
LIN {X 0,Y 254.652,Z 486.629,A -85,B 0,C 180,E1 -715.747,E2 -715.747} C_VEL
LIN {X 0,Y 257.106,Z 492.227,A -85,B 0,C 180,E1 -719.445,E2 -719.445} C_VEL
LIN {X 0,Y 257.783,Z 494.189,A -85,B 0,C 180,E1 -720.356,E2 -720.356} C_VEL
LIN {X 0,Y 246.172,Z 589.584,A -85,B 0,C 180,E1 -721.93,E2 -721.93} C_VEL
LIN {X 0,Y 241.557,Z 611.981,A -85,B 0,C 180,E1 -722.397,E2 -722.397} C_VEL
LIN {X 0,Y 235.344,Z 633.347,A -85,B 0,C 180,E1 -722.924,E2 -722.924} C_VEL
LIN {X 0,Y 227.413,Z 654.585,A -85,B 0,C 180,E1 -723.637,E2 -723.637} C_VEL
LIN {X 0,Y 218.636,Z 673.827,A -85,B 0,C 180,E1 -724.519,E2 -724.519} C_VEL
LIN {X 0,Y 207.993,Z 693.362,A -85,B 0,C 180,E1 -725.719,E2 -725.719} C_VEL
LIN {X 0,Y 196.027,Z 711.88,A -85,B 0,C 180,E1 -727.251,E2 -727.251} C_VEL
LIN {X 0,Y 183.293,Z 728.9,A -85,B 0,C 180,E1 -729.148,E2 -729.148} C_VEL
LIN {X 0,Y 168.88,Z 745.669,A -85,B 0,C 180,E1 -731.708,E2 -731.708} C_VEL
LIN {X 0,Y 162.806,Z 752.126,A -85,B 0,C 180,E1 -732.955,E2 -732.955} C_VEL
LIN {X 0,Y 157.272,Z 757.197,A -85,B 0,C 180,E1 -733.758,E2 -733.758} C_VEL
LIN {X 0,Y 141.286,Z 768.967,A -85,B 0,C 180,E1 -734.942,E2 -734.942} C_VEL
LIN {X 0,Y 135.503,Z 773.384,A -85,B 0,C 180,E1 -736.046,E2 -736.046} C_VEL
LIN {X 0,Y 120.096,Z 785.246,A -85,B 0,C 180,E1 -741.194,E2 -741.194} C_VEL
LIN {X 0,Y 106.094,Z 794.992,A -85,B 0,C 180,E1 -747.653,E2 -747.653} C_VEL
LIN {X 0,Y 92.499,Z 803.828,A -85,B 0,C 180,E1 -756.891,E2 -756.891} C_VEL
LIN {X 0,Y 81.842,Z 810.753,A -85,B 0,C 180,E1 -768.732,E2 -768.732} C_VEL
LIN {X 0,Y 75.139,Z 815.788,A -85,B 0,C 180,E1 -783.109,E2 -783.109} C_VEL
LIN {X 0,Y 72.936,Z 818.971,A -85,B 0,C 180,E1 -798.142,E2 -798.142} C_VEL
LIN {X 0,Y 73.31,Z 820.227,A -85,B 0,C 180,E1 -808.445,E2 -808.445} C_VEL
LIN {X 0,Y 73.028,Z 820.58,A -85,B 0,C 180,E1 -815.508,E2 -815.508} C_VEL
LIN {X 0,Y 73.353,Z 820.153,A -85,B 0,C 180,E1 -829.104,E2 -829.104} C_VEL
LIN {X 0,Y 78.192,Z 818.289,A -85,B 0,C 180,E1 -845.138,E2 -845.138} C_VEL
LIN {X 0,Y 89.005,Z 814.409,A -85,B 0,C 180,E1 -859.818,E2 -859.818} C_VEL
